      MD311 AT %MD311 : UDINT := 16#00000000;  (* RAD[1].Fk: Площадь конвекции *)
      MD312 AT %MD312 : UDINT := 16#00000000;  (* RAD[1].Q0: Расход своб конвекции *)
      MD313 AT %MD313 : UDINT := 16#00000000;  (* RAD[1].Q1: Расход принуд конвекции *)
      MD314 AT %MD314 : UDINT := 16#00000000;  (* RAD[1].Bl[0]: Vобдува- 1 вентилятор *)
      MD315 AT %MD315 : UDINT := 16#00000000;  (* RAD[1].Bl[1]: Vобдува- 2 вентилятора *)
      MD316 AT %MD316 : UDINT := 16#00000000;  (* RAD[1].Bl[2]: Vобдува- 3 вентилятора *)
      MD317 AT %MD317 : UDINT := 16#00000000;  (* RAD[1].Bl[3]: Vобдува- 4 вентилятора *)
      MD318 AT %MD318 : UDINT := 16#00000000;  (* RAD[2].Vm: Объем радиатора *)
      MD319 AT %MD319 : UDINT := 16#00000000;  (* RAD[2].Fk: Площадь конвекции *)
      MD320 AT %MD320 : UDINT := 16#00000000;  (* RAD[2].Q0: Расход своб конвекции *)
      MD321 AT %MD321 : UDINT := 16#00000000;  (* RAD[2].Q1: Расход принуд конвекции *)
      MD322 AT %MD322 : UDINT := 16#00000000;  (* RAD[2].Bl[0]: Vобдува- 1 вентилятор *)
      MD323 AT %MD323 : UDINT := 16#00000000;  (* RAD[2].Bl[1]: Vобдува- 2 вентилятора *)
      MD324 AT %MD324 : UDINT := 16#00000000;  (* RAD[2].Bl[2]: Vобдува- 3 вентилятора *)
      MD325 AT %MD325 : UDINT := 16#00000000;  (* RAD[2].Bl[3]: Vобдува- 4 вентилятора *)
      MD326 AT %MD326 : UDINT := 16#00000000;  (* RAD[3].Vm: Объем радиатора *)
      MD327 AT %MD327 : UDINT := 16#00000000;  (* RAD[3].Fk: Площадь конвекции *)
      MD328 AT %MD328 : UDINT := 16#00000000;  (* RAD[3].Q0: Расход своб конвекции *)
      MD329 AT %MD329 : UDINT := 16#00000000;  (* RAD[3].Q1: Расход принуд конвекции *)
      MD330 AT %MD330 : UDINT := 16#00000000;  (* RAD[3].Bl[0]: Vобдува- 1 вентилятор *)
      MD331 AT %MD331 : UDINT := 16#00000000;  (* RAD[3].Bl[1]: Vобдува- 2 вентилятора *)
      MD332 AT %MD332 : UDINT := 16#00000000;  (* RAD[3].Bl[2]: Vобдува- 3 вентилятора *)
      MD333 AT %MD333 : UDINT := 16#00000000;  (* RAD[3].Bl[3]: Vобдува- 4 вентилятора *)
      MD334 AT %MD334 : UDINT := 16#00000000;  (* RAD[4].Vm: Объем радиатора *)
      MD335 AT %MD335 : UDINT := 16#00000000;  (* RAD[4].Fk: Площадь конвекции *)
      MD336 AT %MD336 : UDINT := 16#00000000;  (* RAD[4].Q0: Расход своб конвекции *)
      MD337 AT %MD337 : UDINT := 16#00000000;  (* RAD[4].Q1: Расход принуд конвекции *)
      MD338 AT %MD338 : UDINT := 16#00000000;  (* RAD[4].Bl[0]: Vобдува- 1 вентилятор *)
      MD339 AT %MD339 : UDINT := 16#00000000;  (* RAD[4].Bl[1]: Vобдува- 2 вентилятора *)
      MD340 AT %MD340 : UDINT := 16#00000000;  (* RAD[4].Bl[2]: Vобдува- 3 вентилятора *)
      MD341 AT %MD341 : UDINT := 16#00000000;  (* RAD[4].Bl[3]: Vобдува- 4 вентилятора *)
      MD342 AT %MD342 : UDINT := 16#00000000;  (* RAD[5].Vm: Объем радиатора *)
      MD343 AT %MD343 : UDINT := 16#00000000;  (* RAD[5].Fk: Площадь конвекции *)
      MD344 AT %MD344 : UDINT := 16#00000000;  (* RAD[5].Q0: Расход своб конвекции *)
      MD345 AT %MD345 : UDINT := 16#00000000;  (* RAD[5].Q1: Расход принуд конвекции *)
      MD346 AT %MD346 : UDINT := 16#00000000;  (* RAD[5].Bl[0]: Vобдува- 1 вентилятор *)
      MD347 AT %MD347 : UDINT := 16#00000000;  (* RAD[5].Bl[1]: Vобдува- 2 вентилятора *)
      MD348 AT %MD348 : UDINT := 16#00000000;  (* RAD[5].Bl[2]: Vобдува- 3 вентилятора *)
      MD349 AT %MD349 : UDINT := 16#00000000;  (* RAD[5].Bl[3]: Vобдува- 4 вентилятора *)
      MD350 AT %MD350 : UDINT := 16#00000000;  (* RAD[6].Vm: Объем радиатора *)
      MD351 AT %MD351 : UDINT := 16#00000000;  (* RAD[6].Fk: Площадь конвекции *)
      MD352 AT %MD352 : UDINT := 16#00000000;  (* RAD[6].Q0: Расход своб конвекции *)
      MD353 AT %MD353 : UDINT := 16#00000000;  (* RAD[6].Q1: Расход принуд конвекции *)
      MD354 AT %MD354 : UDINT := 16#00000000;  (* RAD[6].Bl[0]: Vобдува- 1 вентилятор *)
      MD355 AT %MD355 : UDINT := 16#00000000;  (* RAD[6].Bl[1]: Vобдува- 2 вентилятора *)
      MD356 AT %MD356 : UDINT := 16#00000000;  (* RAD[6].Bl[2]: Vобдува- 3 вентилятора *)
      MD357 AT %MD357 : UDINT := 16#00000000;  (* RAD[6].Bl[3]: Vобдува- 4 вентилятора *)
      MD358 AT %MD358 : UDINT := 16#00000000;  (* RAD[7].Vm: Объем радиатора *)
      MD359 AT %MD359 : UDINT := 16#00000000;  (* RAD[7].Fk: Площадь конвекции *)
      MD360 AT %MD360 : UDINT := 16#00000000;  (* RAD[7].Q0: Расход своб конвекции *)
      MD361 AT %MD361 : UDINT := 16#00000000;  (* RAD[7].Q1: Расход принуд конвекции *)
      MD362 AT %MD362 : UDINT := 16#00000000;  (* RAD[7].Bl[0]: Vобдува- 1 вентилятор *)
      MD363 AT %MD363 : UDINT := 16#00000000;  (* RAD[7].Bl[1]: Vобдува- 2 вентилятора *)
      MD364 AT %MD364 : UDINT := 16#00000000;  (* RAD[7].Bl[2]: Vобдува- 3 вентилятора *)
      MD365 AT %MD365 : UDINT := 16#00000000;  (* RAD[7].Bl[3]: Vобдува- 4 вентилятора *)
      MD366 AT %MD366 : UDINT := 16#00000000;  (* RAD[8].Vm: Объем радиатора *)
      MD367 AT %MD367 : UDINT := 16#00000000;  (* RAD[8].Fk: Площадь конвекции *)
      MD368 AT %MD368 : UDINT := 16#00000000;  (* RAD[8].Q0: Расход своб конвекции *)
      MD369 AT %MD369 : UDINT := 16#00000000;  (* RAD[8].Q1: Расход принуд конвекции *)
      MD370 AT %MD370 : UDINT := 16#00000000;  (* RAD[8].Bl[0]: Vобдува- 1 вентилятор *)
      MD371 AT %MD371 : UDINT := 16#00000000;  (* RAD[8].Bl[1]: Vобдува- 2 вентилятора *)
      MD372 AT %MD372 : UDINT := 16#00000000;  (* RAD[8].Bl[2]: Vобдува- 3 вентилятора *)
      MD373 AT %MD373 : UDINT := 16#00000000;  (* RAD[8].Bl[3]: Vобдува- 4 вентилятора *)
      MD374 AT %MD374 : UDINT := 16#00000000;  (* RAD[9].Vm: Объем радиатора *)
      MD375 AT %MD375 : UDINT := 16#00000000;  (* RAD[9].Fk: Площадь конвекции *)
      MD376 AT %MD376 : UDINT := 16#00000000;  (* RAD[9].Q0: Расход своб конвекции *)
      MD377 AT %MD377 : UDINT := 16#00000000;  (* RAD[9].Q1: Расход принуд конвекции *)
      MD378 AT %MD378 : UDINT := 16#00000000;  (* RAD[9].Bl[0]: Vобдува- 1 вентилятор *)
      MD379 AT %MD379 : UDINT := 16#00000000;  (* RAD[9].Bl[1]: Vобдува- 2 вентилятора *)
      MD380 AT %MD380 : UDINT := 16#00000000;  (* RAD[9].Bl[2]: Vобдува- 3 вентилятора *)
      MD381 AT %MD381 : UDINT := 16#00000000;  (* RAD[9].Bl[3]: Vобдува- 4 вентилятора *)
      MD382 AT %MD382 : UDINT := 16#00000000;  (* RAD[10].Vm: Объем радиатора *)
      MD383 AT %MD383 : UDINT := 16#00000000;  (* RAD[10].Fk: Площадь конвекции *)
      MD384 AT %MD384 : UDINT := 16#00000000;  (* RAD[10].Q0: Расход своб конвекции *)
      MD385 AT %MD385 : UDINT := 16#00000000;  (* RAD[10].Q1: Расход принуд конвекции *)
      MD386 AT %MD386 : UDINT := 16#00000000;  (* RAD[10].Bl[0]: Vобдува- 1 вентилятор *)
      MD387 AT %MD387 : UDINT := 16#00000000;  (* RAD[10].Bl[1]: Vобдува- 2 вентилятора *)
      MD388 AT %MD388 : UDINT := 16#00000000;  (* RAD[10].Bl[2]: Vобдува- 3 вентилятора *)
      MD389 AT %MD389 : UDINT := 16#00000000;  (* RAD[10].Bl[3]: Vобдува- 4 вентилятора *)
      MD390 AT %MD390 : UDINT := 16#00000000;  (* RAD[11].Vm: Объем радиатора *)
      MD391 AT %MD391 : UDINT := 16#00000000;  (* RAD[11].Fk: Площадь конвекции *)
      MD392 AT %MD392 : UDINT := 16#00000000;  (* RAD[11].Q0: Расход своб конвекции *)
      MD393 AT %MD393 : UDINT := 16#00000000;  (* RAD[11].Q1: Расход принуд конвекции *)
      MD394 AT %MD394 : UDINT := 16#00000000;  (* RAD[11].Bl[0]: Vобдува- 1 вентилятор *)
      MD395 AT %MD395 : UDINT := 16#00000000;  (* RAD[11].Bl[1]: Vобдува- 2 вентилятора *)
      MD396 AT %MD396 : UDINT := 16#00000000;  (* RAD[11].Bl[2]: Vобдува- 3 вентилятора *)
      MD397 AT %MD397 : UDINT := 16#00000000;  (* RAD[11].Bl[3]: Vобдува- 4 вентилятора *)
      MD398 AT %MD398 : UDINT := 16#00000000;  (* RAD[12].Vm: Объем радиатора *)
      MD399 AT %MD399 : UDINT := 16#00000000;  (* RAD[12].Fk: Площадь конвекции *)
      MD400 AT %MD400 : UDINT := 16#00000000;  (* RAD[12].Q0: Расход своб конвекции *)
      MD401 AT %MD401 : UDINT := 16#00000000;  (* RAD[12].Q1: Расход принуд конвекции *)
      MD402 AT %MD402 : UDINT := 16#00000000;  (* RAD[12].Bl[0]: Vобдува- 1 вентилятор *)
      MD403 AT %MD403 : UDINT := 16#00000000;  (* RAD[12].Bl[1]: Vобдува- 2 вентилятора *)
      MD404 AT %MD404 : UDINT := 16#00000000;  (* RAD[12].Bl[2]: Vобдува- 3 вентилятора *)
      MD405 AT %MD405 : UDINT := 16#00000000;  (* RAD[12].Bl[3]: Vобдува- 4 вентилятора *)
      MD406 AT %MD406 : UDINT := 16#00000000;  (* RAD[13].Vm: Объем радиатора *)
      MD407 AT %MD407 : UDINT := 16#00000000;  (* RAD[13].Fk: Площадь конвекции *)
      MD408 AT %MD408 : UDINT := 16#00000000;  (* RAD[13].Q0: Расход своб конвекции *)
      MD409 AT %MD409 : UDINT := 16#00000000;  (* RAD[13].Q1: Расход принуд конвекции *)
      MD410 AT %MD410 : UDINT := 16#00000000;  (* RAD[13].Bl[0]: Vобдува- 1 вентилятор *)
      MD411 AT %MD411 : UDINT := 16#00000000;  (* RAD[13].Bl[1]: Vобдува- 2 вентилятора *)
      MD412 AT %MD412 : UDINT := 16#00000000;  (* RAD[13].Bl[2]: Vобдува- 3 вентилятора *)
      MD413 AT %MD413 : UDINT := 16#00000000;  (* RAD[13].Bl[3]: Vобдува- 4 вентилятора *)
      MD414 AT %MD414 : UDINT := 16#00000000;  (* RAD[14].Vm: Объем радиатора *)
      MD415 AT %MD415 : UDINT := 16#00000000;  (* RAD[14].Fk: Площадь конвекции *)
      MD416 AT %MD416 : UDINT := 16#00000000;  (* RAD[14].Q0: Расход своб конвекции *)
      MD417 AT %MD417 : UDINT := 16#00000000;  (* RAD[14].Q1: Расход принуд конвекции *)
      MD418 AT %MD418 : UDINT := 16#00000000;  (* RAD[14].Bl[0]: Vобдува- 1 вентилятор *)
      MD419 AT %MD419 : UDINT := 16#00000000;  (* RAD[14].Bl[1]: Vобдува- 2 вентилятора *)
      MD420 AT %MD420 : UDINT := 16#00000000;  (* RAD[14].Bl[2]: Vобдува- 3 вентилятора *)
      MD421 AT %MD421 : UDINT := 16#00000000;  (* RAD[14].Bl[3]: Vобдува- 4 вентилятора *)
      MD422 AT %MD422 : UDINT := 16#00000000;  (* RAD[15].Vm: Объем радиатора *)
      MD423 AT %MD423 : UDINT := 16#00000000;  (* RAD[15].Fk: Площадь конвекции *)
      MD424 AT %MD424 : UDINT := 16#00000000;  (* RAD[15].Q0: Расход своб конвекции *)
      MD425 AT %MD425 : UDINT := 16#00000000;  (* RAD[15].Q1: Расход принуд конвекции *)
      MD426 AT %MD426 : UDINT := 16#00000000;  (* RAD[15].Bl[0]: Vобдува- 1 вентилятор *)
      MD427 AT %MD427 : UDINT := 16#00000000;  (* RAD[15].Bl[1]: Vобдува- 2 вентилятора *)
      MD428 AT %MD428 : UDINT := 16#00000000;  (* RAD[15].Bl[2]: Vобдува- 3 вентилятора *)
      MD429 AT %MD429 : UDINT := 16#00000000;  (* RAD[15].Bl[3]: Vобдува- 4 вентилятора *)
      MD430 AT %MD430 : UDINT := 16#00000000;  (* HDI.DTI: Дата (секунд от 1970-01-01) *)
      MD431 AT %MD431 : UDINT := 16#00000000;  (* HDI.TMI: Время (милисек с 00:00) *)
      MD432 AT %MD432 : UDINT := 16#00000000;  (* HDI.TOV: Темп. окр. воздуха *)
      MD433 AT %MD433 : UDINT := 16#00000000;  (* HDI.TMH: Темп. верх. слоёв масла *)
      MD434 AT %MD434 : UDINT := 16#00000000;  (* HDI.RVI[0]: Резерв 0 *)
      MD435 AT %MD435 : UDINT := 16#00000000;  (* HDI.RVI[1]: Резерв 1 *)
      MD436 AT %MD436 : UDINT := 16#00000000;  (* PHI[0].Ic: Ток нагрузки *)
      MD437 AT %MD437 : UDINT := 16#00000000;  (* PHI[0].Tin: Т входа из сист.охл. *)
      MD438 AT %MD438 : UDINT := 16#00000000;  (* PHI[0].Tout: Т выхода из сист.охл. *)
      MD439 AT %MD439 : UDINT := 16#00000000;  (* PHI[0].Rn: 32-бит состояния РПН *)
      MD440 AT %MD440 : UDINT := 16#00000000;  (* PHI[0].RD[0,1]: Радиатор-0,1: Тип-Состояние *)
      MD441 AT %MD441 : UDINT := 16#00000000;  (* PHI[0].RD[2,3]: Радиатор-2,3: Тип-Состояние *)
      MD442 AT %MD442 : UDINT := 16#00000000;  (* PHI[0].RD[4,5]: Радиатор-4,5: Тип-Состояние *)
      MD443 AT %MD443 : UDINT := 16#00000000;  (* PHI[0].RD[6,7]: Радиатор-6,7: Тип-Состояние *)
      MD444 AT %MD444 : UDINT := 16#00000000;  (* PHI[1].Ic: Ток нагрузки *)
      MD445 AT %MD445 : UDINT := 16#00000000;  (* PHI[1].Tin: Т входа из сист.охл. *)
      MD446 AT %MD446 : UDINT := 16#00000000;  (* PHI[1].Tout: Т выхода из сист.охл. *)
      MD447 AT %MD447 : UDINT := 16#00000000;  (* PHI[1].Rn: 32-бит состояния РПН *)
      MD448 AT %MD448 : UDINT := 16#00000000;  (* PHI[1].RD[0,1]: Радиатор-0,1: Тип-Состояние *)
      MD449 AT %MD449 : UDINT := 16#00000000;  (* PHI[1].RD[2,3]: Радиатор-2,3: Тип-Состояние *)
      MD450 AT %MD450 : UDINT := 16#00000000;  (* PHI[1].RD[4,5]: Радиатор-4,5: Тип-Состояние *)
      MD451 AT %MD451 : UDINT := 16#00000000;  (* PHI[1].RD[6,7]: Радиатор-6,7: Тип-Состояние *)
      MD452 AT %MD452 : UDINT := 16#00000000;  (* PHI[2].Ic: Ток нагрузки *)
      MD453 AT %MD453 : UDINT := 16#00000000;  (* PHI[2].Tin: Т входа из сист.охл. *)
      MD454 AT %MD454 : UDINT := 16#00000000;  (* PHI[2].Tout: Т выхода из сист.охл. *)
      MD455 AT %MD455 : UDINT := 16#00000000;  (* PHI[2].Rn: 32-бит состояния РПН *)
      MD456 AT %MD456 : UDINT := 16#00000000;  (* PHI[2].RD[0,1]: Радиатор-0,1: Тип-Состояние *)
      MD457 AT %MD457 : UDINT := 16#00000000;  (* PHI[2].RD[2,3]: Радиатор-2,3: Тип-Состояние *)
      MD458 AT %MD458 : UDINT := 16#00000000;  (* PHI[2].RD[4,5]: Радиатор-4,5: Тип-Состояние *)
      MD459 AT %MD459 : UDINT := 16#00000000;  (* PHI[2].RD[6,7]: Радиатор-6,7: Тип-Состояние *)
      MD460 AT %MD460 : UDINT := 16#00000000;  (* HDO.DTO: Дата (секунд от 1970-01-01) *)
      MD461 AT %MD461 : UDINT := 16#00000000;  (* HDO.TMO: Время (милисек с 00:00) *)
      MD462 AT %MD462 : UDINT := 16#00000000;  (* HDO.QTY: Плотность потока ярма *)
      MD463 AT %MD463 : UDINT := 16#00000000;  (* HDO.QTS: Общее тепловыделение *)
      MD464 AT %MD464 : UDINT := 16#00000000;  (* HDO.RVO[0]: Резерв 0 *)
      MD465 AT %MD465 : UDINT := 16#00000000;  (* HDO.RVO[1]: Резерв 1 *)
      MD466 AT %MD466 : UDINT := 16#00000000;  (* PHO[0].Q0: Плотность потока стержня *)
      MD467 AT %MD467 : UDINT := 16#00000000;  (* PHO[0].Q1: Плотность потока обмотки НН *)
      MD468 AT %MD468 : UDINT := 16#00000000;  (* PHO[0].Q2: Плотность потока обмотки ВН *)
      MD469 AT %MD469 : UDINT := 16#00000000;  (* PHO[0].Tin: Т входа из сист.охл. *)
      MD470 AT %MD470 : UDINT := 16#00000000;  (* PHO[0].Tout: Т выхода из сист.охл. *)
      MD471 AT %MD471 : UDINT := 16#00000000;  (* PHO[0].Qm: Суммарный расход масла на фазу *)
      MD472 AT %MD472 : UDINT := 16#00000000;  (* PHO[0].Se: Экв площадь сечения каналов *)
      MD473 AT %MD473 : UDINT := 16#00000000;  (* PHO[0].Ve: Скорость тока масла на фазу *)
      MD474 AT %MD474 : UDINT := 16#00000000;  (* PHO[1].Q0: Плотность потока стержня *)
      MD475 AT %MD475 : UDINT := 16#00000000;  (* PHO[1].Q1: Плотность потока обмотки НН *)
      MD476 AT %MD476 : UDINT := 16#00000000;  (* PHO[1].Q2: Плотность потока обмотки ВН *)
      MD477 AT %MD477 : UDINT := 16#00000000;  (* PHO[1].Tin: Т входа из сист.охл. *)
      MD478 AT %MD478 : UDINT := 16#00000000;  (* PHO[1].Tout: Т выхода из сист.охл. *)
      MD479 AT %MD479 : UDINT := 16#00000000;  (* PHO[1].Qm: Суммарный расход масла на фазу *)
      MD480 AT %MD480 : UDINT := 16#00000000;  (* PHO[1].Se: Экв площадь сечения каналов *)
      MD481 AT %MD481 : UDINT := 16#00000000;  (* PHO[1].Ve: Скорость тока масла на фазу *)
      MD482 AT %MD482 : UDINT := 16#00000000;  (* PHO[2].Q0: Плотность потока стержня *)
      MD483 AT %MD483 : UDINT := 16#00000000;  (* PHO[2].Q1: Плотность потока обмотки НН *)
      MD484 AT %MD484 : UDINT := 16#00000000;  (* PHO[2].Q2: Плотность потока обмотки ВН *)
      MD485 AT %MD485 : UDINT := 16#00000000;  (* PHO[2].Tin: Т входа из сист.охл. *)
      MD486 AT %MD486 : UDINT := 16#00000000;  (* PHO[2].Tout: Т выхода из сист.охл. *)
      MD487 AT %MD487 : UDINT := 16#00000000;  (* PHO[2].Qm: Суммарный расход масла на фазу *)
      MD488 AT %MD488 : UDINT := 16#00000000;  (* PHO[2].Se: Экв площадь сечения каналов *)
      MD489 AT %MD489 : UDINT := 16#00000000;  (* PHO[2].Ve: Скорость тока масла на фазу *)
      MD490 AT %MD490 : UDINT := 16#00000000;  (* RES.DR: Дата (секунд от 1970-01-01) *)
      MD491 AT %MD491 : UDINT := 16#00000000;  (* RES.TR: Время (милисек с 00:00) *)
      MD492 AT %MD492 : UDINT := 16#00000000;  (* RES.FP: Факт. время расчёта (милисек) *)
      MD493 AT %MD493 : UDINT := 16#00000000;  (* RES.ER|RES.FL: Ошибка(UINT)|Флаги(WORD) *)
      MD494 AT %MD494 : UDINT := 16#00000000;  (* RES.RD[0]: Резерв 0 *)
      MD495 AT %MD495 : UDINT := 16#00000000;  (* RES.RD[1]: Резерв 1 *)
      MD496 AT %MD496 : UDINT := 16#00000000;  (* RES.RD[2]: Резерв 2 *)
      MD497 AT %MD497 : UDINT := 16#00000000;  (* RES.RD[3]: Резерв 3 *)
      MD498 AT %MD498 : UDINT := 16#00000000;  (* RES.RD[4]: Резерв 4 *)
      MD499 AT %MD499 : UDINT := 16#00000000;  (* RES.RD[5]: Резерв 5 *)
      MD500 AT %MD500 : UDINT := 16#00000000;  (* CDN[0].(ID|Tmid): Идент.|Tсред. *)
      MD501 AT %MD501 : UDINT := 16#00000000;  (* CDN[0].Tmin.(Ti |XYZ[0]): Темп. |Коорд.X *)
      MD502 AT %MD502 : UDINT := 16#00000000;  (* CDN[0].Tmin.(XYZ[1]|XYZ[2]): Коорд.Y|Коорд.Z *)
      MD503 AT %MD503 : UDINT := 16#00000000;  (* CDN[0].Tmax.(Ti |XYZ[0]): Темп. |Коорд.X *)
      MD504 AT %MD504 : UDINT := 16#00000000;  (* CDN[0].Tmax.(XYZ[1]|XYZ[2]): Коорд.Y|Коорд.Z *)
      MD505 AT %MD505 : UDINT := 16#00000000;  (* CDN[1].(ID|Tmid): Идент.|Tсред. *)
      MD506 AT %MD506 : UDINT := 16#00000000;  (* CDN[1].Tmin.(Ti |XYZ[0]): Темп. |Коорд.X *)
      MD507 AT %MD507 : UDINT := 16#00000000;  (* CDN[1].Tmin.(XYZ[1]|XYZ[2]): Коорд.Y|Коорд.Z *)
      MD508 AT %MD508 : UDINT := 16#00000000;  (* CDN[1].Tmax.(Ti |XYZ[0]): Темп. |Коорд.X *)
      MD509 AT %MD509 : UDINT := 16#00000000;  (* CDN[1].Tmax.(XYZ[1]|XYZ[2]): Коорд.Y|Коорд.Z *)
      MD510 AT %MD510 : UDINT := 16#00000000;  (* CDN[2].(ID|Tmid): Идент.|Tсред. *)
      MD511 AT %MD511 : UDINT := 16#00000000;  (* CDN[2].Tmin.(Ti |XYZ[0]): Темп. |Коорд.X *)
      MD512 AT %MD512 : UDINT := 16#00000000;  (* CDN[2].Tmin.(XYZ[1]|XYZ[2]): Коорд.Y|Коорд.Z *)
      MD513 AT %MD513 : UDINT := 16#00000000;  (* CDN[2].Tmax.(Ti |XYZ[0]): Темп. |Коорд.X *)
      MD514 AT %MD514 : UDINT := 16#00000000;  (* CDN[2].Tmax.(XYZ[1]|XYZ[2]): Коорд.Y|Коорд.Z *)
      MD515 AT %MD515 : UDINT := 16#00000000;  (* CDN[3].(ID|Tmid): Идент.|Tсред. *)
      MD516 AT %MD516 : UDINT := 16#00000000;  (* CDN[3].Tmin.(Ti |XYZ[0]): Темп. |Коорд.X *)
      MD517 AT %MD517 : UDINT := 16#00000000;  (* CDN[3].Tmin.(XYZ[1]|XYZ[2]): Коорд.Y|Коорд.Z *)
      MD518 AT %MD518 : UDINT := 16#00000000;  (* CDN[3].Tmax.(Ti |XYZ[0]): Темп. |Коорд.X *)
      MD519 AT %MD519 : UDINT := 16#00000000;  (* CDN[3].Tmax.(XYZ[1]|XYZ[2]): Коорд.Y|Коорд.Z *)
      MD520 AT %MD520 : UDINT := 16#00000000;  (* CDN[4].(ID|Tmid): Идент.|Tсред. *)
      MD521 AT %MD521 : UDINT := 16#00000000;  (* CDN[4].Tmin.(Ti |XYZ[0]): Темп. |Коорд.X *)
      MD522 AT %MD522 : UDINT := 16#00000000;  (* CDN[4].Tmin.(XYZ[1]|XYZ[2]): Коорд.Y|Коорд.Z *)
      MD523 AT %MD523 : UDINT := 16#00000000;  (* CDN[4].Tmax.(Ti |XYZ[0]): Темп. |Коорд.X *)
      MD524 AT %MD524 : UDINT := 16#00000000;  (* CDN[4].Tmax.(XYZ[1]|XYZ[2]): Коорд.Y|Коорд.Z *)
      MD525 AT %MD525 : UDINT := 16#00000000;  (* CDN[5].(ID|Tmid): Идент.|Tсред. *)
      MD526 AT %MD526 : UDINT := 16#00000000;  (* CDN[5].Tmin.(Ti |XYZ[0]): Темп. |Коорд.X *)
      MD527 AT %MD527 : UDINT := 16#00000000;  (* CDN[5].Tmin.(XYZ[1]|XYZ[2]): Коорд.Y|Коорд.Z *)
      MD528 AT %MD528 : UDINT := 16#00000000;  (* CDN[5].Tmax.(Ti |XYZ[0]): Темп. |Коорд.X *)
      MD529 AT %MD529 : UDINT := 16#00000000;  (* CDN[5].Tmax.(XYZ[1]|XYZ[2]): Коорд.Y|Коорд.Z *)
      MD530 AT %MD530 : UDINT := 16#00000000;  (* CDN[6].(ID|Tmid): Идент.|Tсред. *)
      MD531 AT %MD531 : UDINT := 16#00000000;  (* CDN[6].Tmin.(Ti |XYZ[0]): Темп. |Коорд.X *)
      MD532 AT %MD532 : UDINT := 16#00000000;  (* CDN[6].Tmin.(XYZ[1]|XYZ[2]): Коорд.Y|Коорд.Z *)
      MD533 AT %MD533 : UDINT := 16#00000000;  (* CDN[6].Tmax.(Ti |XYZ[0]): Темп. |Коорд.X *)
      MD534 AT %MD534 : UDINT := 16#00000000;  (* CDN[6].Tmax.(XYZ[1]|XYZ[2]): Коорд.Y|Коорд.Z *)
      MD535 AT %MD535 : UDINT := 16#00000000;  (* CDN[7].(ID|Tmid): Идент.|Tсред. *)
      MD536 AT %MD536 : UDINT := 16#00000000;  (* CDN[7].Tmin.(Ti |XYZ[0]): Темп. |Коорд.X *)
      MD537 AT %MD537 : UDINT := 16#00000000;  (* CDN[7].Tmin.(XYZ[1]|XYZ[2]): Коорд.Y|Коорд.Z *)
      MD538 AT %MD538 : UDINT := 16#00000000;  (* CDN[7].Tmax.(Ti |XYZ[0]): Темп. |Коорд.X *)
      MD539 AT %MD539 : UDINT := 16#00000000;  (* CDN[7].Tmax.(XYZ[1]|XYZ[2]): Коорд.Y|Коорд.Z *)
      MD540 AT %MD540 : UDINT := 16#00000000;  (* CDN[8].(ID|Tmid): Идент.|Tсред. *)
      MD541 AT %MD541 : UDINT := 16#00000000;  (* CDN[8].Tmin.(Ti |XYZ[0]): Темп. |Коорд.X *)
      MD542 AT %MD542 : UDINT := 16#00000000;  (* CDN[8].Tmin.(XYZ[1]|XYZ[2]): Коорд.Y|Коорд.Z *)
      MD543 AT %MD543 : UDINT := 16#00000000;  (* CDN[8].Tmax.(Ti |XYZ[0]): Темп. |Коорд.X *)
      MD544 AT %MD544 : UDINT := 16#00000000;  (* CDN[8].Tmax.(XYZ[1]|XYZ[2]): Коорд.Y|Коорд.Z *)
      MD545 AT %MD545 : UDINT := 16#00000000;  (* CDN[9].(ID|Tmid): Идент.|Tсред. *)
      MD546 AT %MD546 : UDINT := 16#00000000;  (* CDN[9].Tmin.(Ti |XYZ[0]): Темп. |Коорд.X *)
      MD547 AT %MD547 : UDINT := 16#00000000;  (* CDN[9].Tmin.(XYZ[1]|XYZ[2]): Коорд.Y|Коорд.Z *)
      MD548 AT %MD548 : UDINT := 16#00000000;  (* CDN[9].Tmax.(Ti |XYZ[0]): Темп. |Коорд.X *)
      MD549 AT %MD549 : UDINT := 16#00000000;  (* CDN[9].Tmax.(XYZ[1]|XYZ[2]): Коорд.Y|Коорд.Z *)
      MD550 AT %MD550 : UDINT := 16#00000000;  (* CDN[10].(ID|Tmid): Идент.|Tсред. *)
      MD551 AT %MD551 : UDINT := 16#00000000;  (* CDN[10].Tmin.(Ti |XYZ[0]): Темп. |Коорд.X *)
      MD552 AT %MD552 : UDINT := 16#00000000;  (* CDN[10].Tmin.(XYZ[1]|XYZ[2]): Коорд.Y|Коорд.Z *)
      MD553 AT %MD553 : UDINT := 16#00000000;  (* CDN[10].Tmax.(Ti |XYZ[0]): Темп. |Коорд.X *)
      MD554 AT %MD554 : UDINT := 16#00000000;  (* CDN[10].Tmax.(XYZ[1]|XYZ[2]): Коорд.Y|Коорд.Z *)
      MD555 AT %MD555 : UDINT := 16#00000000;  (* CDN[11].(ID|Tmid): Идент.|Tсред. *)
      MD556 AT %MD556 : UDINT := 16#00000000;  (* CDN[11].Tmin.(Ti |XYZ[0]): Темп. |Коорд.X *)
      MD557 AT %MD557 : UDINT := 16#00000000;  (* CDN[11].Tmin.(XYZ[1]|XYZ[2]): Коорд.Y|Коорд.Z *)
      MD558 AT %MD558 : UDINT := 16#00000000;  (* CDN[11].Tmax.(Ti |XYZ[0]): Темп. |Коорд.X *)
      MD559 AT %MD559 : UDINT := 16#00000000;  (* CDN[11].Tmax.(XYZ[1]|XYZ[2]): Коорд.Y|Коорд.Z *)
      MD560 AT %MD560 : UDINT := 16#00000000;  (* CDN[12].(ID|Tmid): Идент.|Tсред. *)
      MD561 AT %MD561 : UDINT := 16#00000000;  (* CDN[12].Tmin.(Ti |XYZ[0]): Темп. |Коорд.X *)
      MD562 AT %MD562 : UDINT := 16#00000000;  (* CDN[12].Tmin.(XYZ[1]|XYZ[2]): Коорд.Y|Коорд.Z *)
      MD563 AT %MD563 : UDINT := 16#00000000;  (* CDN[12].Tmax.(Ti |XYZ[0]): Темп. |Коорд.X *)
      MD564 AT %MD564 : UDINT := 16#00000000;  (* CDN[12].Tmax.(XYZ[1]|XYZ[2]): Коорд.Y|Коорд.Z *)
      MD565 AT %MD565 : UDINT := 16#00000000;  (* CDN[13].(ID|Tmid): Идент.|Tсред. *)
      MD566 AT %MD566 : UDINT := 16#00000000;  (* CDN[13].Tmin.(Ti |XYZ[0]): Темп. |Коорд.X *)
      MD567 AT %MD567 : UDINT := 16#00000000;  (* CDN[13].Tmin.(XYZ[1]|XYZ[2]): Коорд.Y|Коорд.Z *)
      MD568 AT %MD568 : UDINT := 16#00000000;  (* CDN[13].Tmax.(Ti |XYZ[0]): Темп. |Коорд.X *)
      MD569 AT %MD569 : UDINT := 16#00000000;  (* CDN[13].Tmax.(XYZ[1]|XYZ[2]): Коорд.Y|Коорд.Z *)
      MD570 AT %MD570 : UDINT := 16#00000000;  (* CDN[14].(ID|Tmid): Идент.|Tсред. *)
      MD571 AT %MD571 : UDINT := 16#00000000;  (* CDN[14].Tmin.(Ti |XYZ[0]): Темп. |Коорд.X *)
      MD572 AT %MD572 : UDINT := 16#00000000;  (* CDN[14].Tmin.(XYZ[1]|XYZ[2]): Коорд.Y|Коорд.Z *)
      MD573 AT %MD573 : UDINT := 16#00000000;  (* CDN[14].Tmax.(Ti |XYZ[0]): Темп. |Коорд.X *)
      MD574 AT %MD574 : UDINT := 16#00000000;  (* CDN[14].Tmax.(XYZ[1]|XYZ[2]): Коорд.Y|Коорд.Z *)
      MD575 AT %MD575 : UDINT := 16#00000000;  (* CDN[15].(ID|Tmid): Идент.|Tсред. *)
      MD576 AT %MD576 : UDINT := 16#00000000;  (* CDN[15].Tmin.(Ti |XYZ[0]): Темп. |Коорд.X *)
      MD577 AT %MD577 : UDINT := 16#00000000;  (* CDN[15].Tmin.(XYZ[1]|XYZ[2]): Коорд.Y|Коорд.Z *)
      MD578 AT %MD578 : UDINT := 16#00000000;  (* CDN[15].Tmax.(Ti |XYZ[0]): Темп. |Коорд.X *)
      MD579 AT %MD579 : UDINT := 16#00000000;  (* CDN[15].Tmax.(XYZ[1]|XYZ[2]): Коорд.Y|Коорд.Z *)
      MD580 AT %MD580 : UDINT := 16#00000000;  (* CDN[16].(ID|Tmid): Идент.|Tсред. *)
      MD581 AT %MD581 : UDINT := 16#00000000;  (* CDN[16].Tmin.(Ti |XYZ[0]): Темп. |Коорд.X *)
      MD582 AT %MD582 : UDINT := 16#00000000;  (* CDN[16].Tmin.(XYZ[1]|XYZ[2]): Коорд.Y|Коорд.Z *)
      MD583 AT %MD583 : UDINT := 16#00000000;  (* CDN[16].Tmax.(Ti |XYZ[0]): Темп. |Коорд.X *)
      MD584 AT %MD584 : UDINT := 16#00000000;  (* CDN[16].Tmax.(XYZ[1]|XYZ[2]): Коорд.Y|Коорд.Z *)
      MD585 AT %MD585 : UDINT := 16#00000000;  (* CDN[17].(ID|Tmid): Идент.|Tсред. *)
      MD586 AT %MD586 : UDINT := 16#00000000;  (* CDN[17].Tmin.(Ti |XYZ[0]): Темп. |Коорд.X *)
      MD587 AT %MD587 : UDINT := 16#00000000;  (* CDN[17].Tmin.(XYZ[1]|XYZ[2]): Коорд.Y|Коорд.Z *)
      MD588 AT %MD588 : UDINT := 16#00000000;  (* CDN[17].Tmax.(Ti |XYZ[0]): Темп. |Коорд.X *)
      MD589 AT %MD589 : UDINT := 16#00000000;  (* CDN[17].Tmax.(XYZ[1]|XYZ[2]): Коорд.Y|Коорд.Z *)
      MD590 AT %MD590 : UDINT := 16#00000000;  (* CDN[18].(ID|Tmid): Идент.|Tсред. *)
      MD591 AT %MD591 : UDINT := 16#00000000;  (* CDN[18].Tmin.(Ti |XYZ[0]): Темп. |Коорд.X *)
      MD592 AT %MD592 : UDINT := 16#00000000;  (* CDN[18].Tmin.(XYZ[1]|XYZ[2]): Коорд.Y|Коорд.Z *)
      MD593 AT %MD593 : UDINT := 16#00000000;  (* CDN[18].Tmax.(Ti |XYZ[0]): Темп. |Коорд.X *)
      MD594 AT %MD594 : UDINT := 16#00000000;  (* CDN[18].Tmax.(XYZ[1]|XYZ[2]): Коорд.Y|Коорд.Z *)
      MD595 AT %MD595 : UDINT := 16#00000000;  (* CDN[19].(ID|Tmid): Идент.|Tсред. *)
      MD596 AT %MD596 : UDINT := 16#00000000;  (* CDN[19].Tmin.(Ti |XYZ[0]): Темп. |Коорд.X *)
      MD597 AT %MD597 : UDINT := 16#00000000;  (* CDN[19].Tmin.(XYZ[1]|XYZ[2]): Коорд.Y|Коорд.Z *)
      MD598 AT %MD598 : UDINT := 16#00000000;  (* CDN[19].Tmax.(Ti |XYZ[0]): Темп. |Коорд.X *)
      MD599 AT %MD599 : UDINT := 16#00000000;  (* CDN[19].Tmax.(XYZ[1]|XYZ[2]): Коорд.Y|Коорд.Z *)
      MD600 AT %MD600 : UDINT := 16#00000000;  (* CDN[20].(ID|Tmid): Идент.|Tсред. *)
      MD601 AT %MD601 : UDINT := 16#00000000;  (* CDN[20].Tmin.(Ti |XYZ[0]): Темп. |Коорд.X *)
      MD602 AT %MD602 : UDINT := 16#00000000;  (* CDN[20].Tmin.(XYZ[1]|XYZ[2]): Коорд.Y|Коорд.Z *)
      MD603 AT %MD603 : UDINT := 16#00000000;  (* CDN[20].Tmax.(Ti |XYZ[0]): Темп. |Коорд.X *)
      MD604 AT %MD604 : UDINT := 16#00000000;  (* CDN[20].Tmax.(XYZ[1]|XYZ[2]): Коорд.Y|Коорд.Z *)
      MD605 AT %MD605 : UDINT := 16#00000000;  (* CDN[21].(ID|Tmid): Идент.|Tсред. *)
      MD606 AT %MD606 : UDINT := 16#00000000;  (* CDN[21].Tmin.(Ti |XYZ[0]): Темп. |Коорд.X *)
      MD607 AT %MD607 : UDINT := 16#00000000;  (* CDN[21].Tmin.(XYZ[1]|XYZ[2]): Коорд.Y|Коорд.Z *)
      MD608 AT %MD608 : UDINT := 16#00000000;  (* CDN[21].Tmax.(Ti |XYZ[0]): Темп. |Коорд.X *)
      MD609 AT %MD609 : UDINT := 16#00000000;  (* CDN[21].Tmax.(XYZ[1]|XYZ[2]): Коорд.Y|Коорд.Z *)
      MD610 AT %MD610 : UDINT := 16#00000000;  (* CDN[22].(ID|Tmid): Идент.|Tсред. *)
      MD611 AT %MD611 : UDINT := 16#00000000;  (* CDN[22].Tmin.(Ti |XYZ[0]): Темп. |Коорд.X *)
      MD612 AT %MD612 : UDINT := 16#00000000;  (* CDN[22].Tmin.(XYZ[1]|XYZ[2]): Коорд.Y|Коорд.Z *)
      MD613 AT %MD613 : UDINT := 16#00000000;  (* CDN[22].Tmax.(Ti |XYZ[0]): Темп. |Коорд.X *)
      MD614 AT %MD614 : UDINT := 16#00000000;  (* CDN[22].Tmax.(XYZ[1]|XYZ[2]): Коорд.Y|Коорд.Z *)
      MD615 AT %MD615 : UDINT := 16#00000000;  (* CDN[23].(ID|Tmid): Идент.|Tсред. *)
      MD616 AT %MD616 : UDINT := 16#00000000;  (* CDN[23].Tmin.(Ti |XYZ[0]): Темп. |Коорд.X *)
      MD617 AT %MD617 : UDINT := 16#00000000;  (* CDN[23].Tmin.(XYZ[1]|XYZ[2]): Коорд.Y|Коорд.Z *)
      MD618 AT %MD618 : UDINT := 16#00000000;  (* CDN[23].Tmax.(Ti |XYZ[0]): Темп. |Коорд.X *)
      MD619 AT %MD619 : UDINT := 16#00000000;  (* CDN[23].Tmax.(XYZ[1]|XYZ[2]): Коорд.Y|Коорд.Z *)
      MD620 AT %MD620 : UDINT := 16#00000000;  (* CDN[24].(ID|Tmid): Идент.|Tсред. *)
      MD621 AT %MD621 : UDINT := 16#00000000;  (* CDN[24].Tmin.(Ti |XYZ[0]): Темп. |Коорд.X *)
      MD622 AT %MD622 : UDINT := 16#00000000;  (* CDN[24].Tmin.(XYZ[1]|XYZ[2]): Коорд.Y|Коорд.Z *)
      MD623 AT %MD623 : UDINT := 16#00000000;  (* CDN[24].Tmax.(Ti |XYZ[0]): Темп. |Коорд.X *)
      MD624 AT %MD624 : UDINT := 16#00000000;  (* CDN[24].Tmax.(XYZ[1]|XYZ[2]): Коорд.Y|Коорд.Z *)
      MD625 AT %MD625 : UDINT := 16#00000000;  (* CDN[25].(ID|Tmid): Идент.|Tсред. *)
      MD626 AT %MD626 : UDINT := 16#00000000;  (* CDN[25].Tmin.(Ti |XYZ[0]): Темп. |Коорд.X *)
      MD627 AT %MD627 : UDINT := 16#00000000;  (* CDN[25].Tmin.(XYZ[1]|XYZ[2]): Коорд.Y|Коорд.Z *)
      MD628 AT %MD628 : UDINT := 16#00000000;  (* CDN[25].Tmax.(Ti |XYZ[0]): Темп. |Коорд.X *)
      MD629 AT %MD629 : UDINT := 16#00000000;  (* CDN[25].Tmax.(XYZ[1]|XYZ[2]): Коорд.Y|Коорд.Z *)
      MD630 AT %MD630 : UDINT := 16#00000000;  (* CDN[26].(ID|Tmid): Идент.|Tсред. *)
      MD631 AT %MD631 : UDINT := 16#00000000;  (* CDN[26].Tmin.(Ti |XYZ[0]): Темп. |Коорд.X *)
      MD632 AT %MD632 : UDINT := 16#00000000;  (* CDN[26].Tmin.(XYZ[1]|XYZ[2]): Коорд.Y|Коорд.Z *)
      MD633 AT %MD633 : UDINT := 16#00000000;  (* CDN[26].Tmax.(Ti |XYZ[0]): Темп. |Коорд.X *)
      MD634 AT %MD634 : UDINT := 16#00000000;  (* CDN[26].Tmax.(XYZ[1]|XYZ[2]): Коорд.Y|Коорд.Z *)
      MD635 AT %MD635 : UDINT := 16#00000000;  (* CDN[27].(ID|Tmid): Идент.|Tсред. *)
      MD636 AT %MD636 : UDINT := 16#00000000;  (* CDN[27].Tmin.(Ti |XYZ[0]): Темп. |Коорд.X *)
      MD637 AT %MD637 : UDINT := 16#00000000;  (* CDN[27].Tmin.(XYZ[1]|XYZ[2]): Коорд.Y|Коорд.Z *)
      MD638 AT %MD638 : UDINT := 16#00000000;  (* CDN[27].Tmax.(Ti |XYZ[0]): Темп. |Коорд.X *)
      MD639 AT %MD639 : UDINT := 16#00000000;  (* CDN[27].Tmax.(XYZ[1]|XYZ[2]): Коорд.Y|Коорд.Z *)
      MD640 AT %MD640 : UDINT := 16#00000000;  (* CDN[28].(ID|Tmid): Идент.|Tсред. *)
      MD641 AT %MD641 : UDINT := 16#00000000;  (* CDN[28].Tmin.(Ti |XYZ[0]): Темп. |Коорд.X *)
      MD642 AT %MD642 : UDINT := 16#00000000;  (* CDN[28].Tmin.(XYZ[1]|XYZ[2]): Коорд.Y|Коорд.Z *)
      MD643 AT %MD643 : UDINT := 16#00000000;  (* CDN[28].Tmax.(Ti |XYZ[0]): Темп. |Коорд.X *)
      MD644 AT %MD644 : UDINT := 16#00000000;  (* CDN[28].Tmax.(XYZ[1]|XYZ[2]): Коорд.Y|Коорд.Z *)
      MD645 AT %MD645 : UDINT := 16#00000000;  (* CDN[29].(ID|Tmid): Идент.|Tсред. *)
      MD646 AT %MD646 : UDINT := 16#00000000;  (* CDN[29].Tmin.(Ti |XYZ[0]): Темп. |Коорд.X *)
      MD647 AT %MD647 : UDINT := 16#00000000;  (* CDN[29].Tmin.(XYZ[1]|XYZ[2]): Коорд.Y|Коорд.Z *)
      MD648 AT %MD648 : UDINT := 16#00000000;  (* CDN[29].Tmax.(Ti |XYZ[0]): Темп. |Коорд.X *)
      MD649 AT %MD649 : UDINT := 16#00000000;  (* CDN[29].Tmax.(XYZ[1]|XYZ[2]): Коорд.Y|Коорд.Z *)
      MD650 AT %MD650 : UDINT := 16#00000000;  (* CDN[30].(ID|Tmid): Идент.|Tсред. *)
      MD651 AT %MD651 : UDINT := 16#00000000;  (* CDN[30].Tmin.(Ti |XYZ[0]): Темп. |Коорд.X *)
      MD652 AT %MD652 : UDINT := 16#00000000;  (* CDN[30].Tmin.(XYZ[1]|XYZ[2]): Коорд.Y|Коорд.Z *)
      MD653 AT %MD653 : UDINT := 16#00000000;  (* CDN[30].Tmax.(Ti |XYZ[0]): Темп. |Коорд.X *)
      MD654 AT %MD654 : UDINT := 16#00000000;  (* CDN[30].Tmax.(XYZ[1]|XYZ[2]): Коорд.Y|Коорд.Z *)
      MD655 AT %MD655 : UDINT := 16#00000000;  (* CDN[31].(ID|Tmid): Идент.|Tсред. *)
      MD656 AT %MD656 : UDINT := 16#00000000;  (* CDN[31].Tmin.(Ti |XYZ[0]): Темп. |Коорд.X *)
      MD657 AT %MD657 : UDINT := 16#00000000;  (* CDN[31].Tmin.(XYZ[1]|XYZ[2]): Коорд.Y|Коорд.Z *)
      MD658 AT %MD658 : UDINT := 16#00000000;  (* CDN[31].Tmax.(Ti |XYZ[0]): Темп. |Коорд.X *)
      MD659 AT %MD659 : UDINT := 16#00000000;  (* CDN[31].Tmax.(XYZ[1]|XYZ[2]): Коорд.Y|Коорд.Z *)
      MD660 AT %MD660 : UDINT := 16#00000000;  (* CDN[32].(ID|Tmid): Идент.|Tсред. *)
      MD661 AT %MD661 : UDINT := 16#00000000;  (* CDN[32].Tmin.(Ti |XYZ[0]): Темп. |Коорд.X *)
      MD662 AT %MD662 : UDINT := 16#00000000;  (* CDN[32].Tmin.(XYZ[1]|XYZ[2]): Коорд.Y|Коорд.Z *)
      MD663 AT %MD663 : UDINT := 16#00000000;  (* CDN[32].Tmax.(Ti |XYZ[0]): Темп. |Коорд.X *)
      MD664 AT %MD664 : UDINT := 16#00000000;  (* CDN[32].Tmax.(XYZ[1]|XYZ[2]): Коорд.Y|Коорд.Z *)
      MD665 AT %MD665 : UDINT := 16#00000000;  (* CDN[33].(ID|Tmid): Идент.|Tсред. *)
      MD666 AT %MD666 : UDINT := 16#00000000;  (* CDN[33].Tmin.(Ti |XYZ[0]): Темп. |Коорд.X *)
      MD667 AT %MD667 : UDINT := 16#00000000;  (* CDN[33].Tmin.(XYZ[1]|XYZ[2]): Коорд.Y|Коорд.Z *)
      MD668 AT %MD668 : UDINT := 16#00000000;  (* CDN[33].Tmax.(Ti |XYZ[0]): Темп. |Коорд.X *)
      MD669 AT %MD669 : UDINT := 16#00000000;  (* CDN[33].Tmax.(XYZ[1]|XYZ[2]): Коорд.Y|Коорд.Z *)
      MD670 AT %MD670 : UDINT := 16#00000000;  (* CDN[34].(ID|Tmid): Идент.|Tсред. *)
      MD671 AT %MD671 : UDINT := 16#00000000;  (* CDN[34].Tmin.(Ti |XYZ[0]): Темп. |Коорд.X *)
      MD672 AT %MD672 : UDINT := 16#00000000;  (* CDN[34].Tmin.(XYZ[1]|XYZ[2]): Коорд.Y|Коорд.Z *)
      MD673 AT %MD673 : UDINT := 16#00000000;  (* CDN[34].Tmax.(Ti |XYZ[0]): Темп. |Коорд.X *)
      MD674 AT %MD674 : UDINT := 16#00000000;  (* CDN[34].Tmax.(XYZ[1]|XYZ[2]): Коорд.Y|Коорд.Z *)
      MD675 AT %MD675 : UDINT := 16#00000000;  (* CDN[35].(ID|Tmid): Идент.|Tсред. *)
      MD676 AT %MD676 : UDINT := 16#00000000;  (* CDN[35].Tmin.(Ti |XYZ[0]): Темп. |Коорд.X *)
      MD677 AT %MD677 : UDINT := 16#00000000;  (* CDN[35].Tmin.(XYZ[1]|XYZ[2]): Коорд.Y|Коорд.Z *)
      MD678 AT %MD678 : UDINT := 16#00000000;  (* CDN[35].Tmax.(Ti |XYZ[0]): Темп. |Коорд.X *)
      MD679 AT %MD679 : UDINT := 16#00000000;  (* CDN[35].Tmax.(XYZ[1]|XYZ[2]): Коорд.Y|Коорд.Z *)
      MD680 AT %MD680 : UDINT := 16#00000000;  (* CDN[36].(ID|Tmid): Идент.|Tсред. *)
      MD681 AT %MD681 : UDINT := 16#00000000;  (* CDN[36].Tmin.(Ti |XYZ[0]): Темп. |Коорд.X *)
      MD682 AT %MD682 : UDINT := 16#00000000;  (* CDN[36].Tmin.(XYZ[1]|XYZ[2]): Коорд.Y|Коорд.Z *)
      MD683 AT %MD683 : UDINT := 16#00000000;  (* CDN[36].Tmax.(Ti |XYZ[0]): Темп. |Коорд.X *)
      MD684 AT %MD684 : UDINT := 16#00000000;  (* CDN[36].Tmax.(XYZ[1]|XYZ[2]): Коорд.Y|Коорд.Z *)
      MD685 AT %MD685 : UDINT := 16#00000000;  (* CDN[37].(ID|Tmid): Идент.|Tсред. *)
      MD686 AT %MD686 : UDINT := 16#00000000;  (* CDN[37].Tmin.(Ti |XYZ[0]): Темп. |Коорд.X *)
      MD687 AT %MD687 : UDINT := 16#00000000;  (* CDN[37].Tmin.(XYZ[1]|XYZ[2]): Коорд.Y|Коорд.Z *)
      MD688 AT %MD688 : UDINT := 16#00000000;  (* CDN[37].Tmax.(Ti |XYZ[0]): Темп. |Коорд.X *)
      MD689 AT %MD689 : UDINT := 16#00000000;  (* CDN[37].Tmax.(XYZ[1]|XYZ[2]): Коорд.Y|Коорд.Z *)
      MD690 AT %MD690 : UDINT := 16#00000000;  (* CDN[38].(ID|Tmid): Идент.|Tсред. *)
      MD691 AT %MD691 : UDINT := 16#00000000;  (* CDN[38].Tmin.(Ti |XYZ[0]): Темп. |Коорд.X *)
      MD692 AT %MD692 : UDINT := 16#00000000;  (* CDN[38].Tmin.(XYZ[1]|XYZ[2]): Коорд.Y|Коорд.Z *)
      MD693 AT %MD693 : UDINT := 16#00000000;  (* CDN[38].Tmax.(Ti |XYZ[0]): Темп. |Коорд.X *)
      MD694 AT %MD694 : UDINT := 16#00000000;  (* CDN[38].Tmax.(XYZ[1]|XYZ[2]): Коорд.Y|Коорд.Z *)
      MD695 AT %MD695 : UDINT := 16#00000000;  (* CDN[39].(ID|Tmid): Идент.|Tсред. *)
      MD696 AT %MD696 : UDINT := 16#00000000;  (* CDN[39].Tmin.(Ti |XYZ[0]): Темп. |Коорд.X *)
      MD697 AT %MD697 : UDINT := 16#00000000;  (* CDN[39].Tmin.(XYZ[1]|XYZ[2]): Коорд.Y|Коорд.Z *)
      MD698 AT %MD698 : UDINT := 16#00000000;  (* CDN[39].Tmax.(Ti |XYZ[0]): Темп. |Коорд.X *)
      MD699 AT %MD699 : UDINT := 16#00000000;  (* CDN[39].Tmax.(XYZ[1]|XYZ[2]): Коорд.Y|Коорд.Z *)
      MD700 AT %MD700 : UDINT := 16#00000000;  (* CDN[40].(ID|Tmid): Идент.|Tсред. *)
      MD701 AT %MD701 : UDINT := 16#00000000;  (* CDN[40].Tmin.(Ti |XYZ[0]): Темп. |Коорд.X *)
      MD702 AT %MD702 : UDINT := 16#00000000;  (* CDN[40].Tmin.(XYZ[1]|XYZ[2]): Коорд.Y|Коорд.Z *)
      MD703 AT %MD703 : UDINT := 16#00000000;  (* CDN[40].Tmax.(Ti |XYZ[0]): Темп. |Коорд.X *)
      MD704 AT %MD704 : UDINT := 16#00000000;  (* CDN[40].Tmax.(XYZ[1]|XYZ[2]): Коорд.Y|Коорд.Z *)
      MD705 AT %MD705 : UDINT := 16#00000000;  (* CDN[41].(ID|Tmid): Идент.|Tсред. *)
      MD706 AT %MD706 : UDINT := 16#00000000;  (* CDN[41].Tmin.(Ti |XYZ[0]): Темп. |Коорд.X *)
      MD707 AT %MD707 : UDINT := 16#00000000;  (* CDN[41].Tmin.(XYZ[1]|XYZ[2]): Коорд.Y|Коорд.Z *)
      MD708 AT %MD708 : UDINT := 16#00000000;  (* CDN[41].Tmax.(Ti |XYZ[0]): Темп. |Коорд.X *)
      MD709 AT %MD709 : UDINT := 16#00000000;  (* CDN[41].Tmax.(XYZ[1]|XYZ[2]): Коорд.Y|Коорд.Z *)
      MD710 AT %MD710 : UDINT := 16#00000000;  (* CDN[42].(ID|Tmid): Идент.|Tсред. *)
      MD711 AT %MD711 : UDINT := 16#00000000;  (* CDN[42].Tmin.(Ti |XYZ[0]): Темп. |Коорд.X *)
      MD712 AT %MD712 : UDINT := 16#00000000;  (* CDN[42].Tmin.(XYZ[1]|XYZ[2]): Коорд.Y|Коорд.Z *)
      MD713 AT %MD713 : UDINT := 16#00000000;  (* CDN[42].Tmax.(Ti |XYZ[0]): Темп. |Коорд.X *)
      MD714 AT %MD714 : UDINT := 16#00000000;  (* CDN[42].Tmax.(XYZ[1]|XYZ[2]): Коорд.Y|Коорд.Z *)
      MD715 AT %MD715 : UDINT := 16#00000000;  (* CDN[43].(ID|Tmid): Идент.|Tсред. *)
      MD716 AT %MD716 : UDINT := 16#00000000;  (* CDN[43].Tmin.(Ti |XYZ[0]): Темп. |Коорд.X *)
      MD717 AT %MD717 : UDINT := 16#00000000;  (* CDN[43].Tmin.(XYZ[1]|XYZ[2]): Коорд.Y|Коорд.Z *)
      MD718 AT %MD718 : UDINT := 16#00000000;  (* CDN[43].Tmax.(Ti |XYZ[0]): Темп. |Коорд.X *)
      MD719 AT %MD719 : UDINT := 16#00000000;  (* CDN[43].Tmax.(XYZ[1]|XYZ[2]): Коорд.Y|Коорд.Z *)
      MD720 AT %MD720 : UDINT := 16#00000000;  (* CDN[44].(ID|Tmid): Идент.|Tсред. *)
      MD721 AT %MD721 : UDINT := 16#00000000;  (* CDN[44].Tmin.(Ti |XYZ[0]): Темп. |Коорд.X *)
      MD722 AT %MD722 : UDINT := 16#00000000;  (* CDN[44].Tmin.(XYZ[1]|XYZ[2]): Коорд.Y|Коорд.Z *)
      MD723 AT %MD723 : UDINT := 16#00000000;  (* CDN[44].Tmax.(Ti |XYZ[0]): Темп. |Коорд.X *)
      MD724 AT %MD724 : UDINT := 16#00000000;  (* CDN[44].Tmax.(XYZ[1]|XYZ[2]): Коорд.Y|Коорд.Z *)
      MD725 AT %MD725 : UDINT := 16#00000000;  (* CDN[45].(ID|Tmid): Идент.|Tсред. *)
      MD726 AT %MD726 : UDINT := 16#00000000;  (* CDN[45].Tmin.(Ti |XYZ[0]): Темп. |Коорд.X *)
      MD727 AT %MD727 : UDINT := 16#00000000;  (* CDN[45].Tmin.(XYZ[1]|XYZ[2]): Коорд.Y|Коорд.Z *)
      MD728 AT %MD728 : UDINT := 16#00000000;  (* CDN[45].Tmax.(Ti |XYZ[0]): Темп. |Коорд.X *)
      MD729 AT %MD729 : UDINT := 16#00000000;  (* CDN[45].Tmax.(XYZ[1]|XYZ[2]): Коорд.Y|Коорд.Z *)
      MD730 AT %MD730 : UDINT := 16#00000000;  (* CDN[46].(ID|Tmid): Идент.|Tсред. *)
      MD731 AT %MD731 : UDINT := 16#00000000;  (* CDN[46].Tmin.(Ti |XYZ[0]): Темп. |Коорд.X *)
      MD732 AT %MD732 : UDINT := 16#00000000;  (* CDN[46].Tmin.(XYZ[1]|XYZ[2]): Коорд.Y|Коорд.Z *)
      MD733 AT %MD733 : UDINT := 16#00000000;  (* CDN[46].Tmax.(Ti |XYZ[0]): Темп. |Коорд.X *)
      MD734 AT %MD734 : UDINT := 16#00000000;  (* CDN[46].Tmax.(XYZ[1]|XYZ[2]): Коорд.Y|Коорд.Z *)
      MD735 AT %MD735 : UDINT := 16#00000000;  (* CDN[47].(ID|Tmid): Идент.|Tсред. *)
      MD736 AT %MD736 : UDINT := 16#00000000;  (* CDN[47].Tmin.(Ti |XYZ[0]): Темп. |Коорд.X *)
      MD737 AT %MD737 : UDINT := 16#00000000;  (* CDN[47].Tmin.(XYZ[1]|XYZ[2]): Коорд.Y|Коорд.Z *)
      MD738 AT %MD738 : UDINT := 16#00000000;  (* CDN[47].Tmax.(Ti |XYZ[0]): Темп. |Коорд.X *)
      MD739 AT %MD739 : UDINT := 16#00000000;  (* CDN[47].Tmax.(XYZ[1]|XYZ[2]): Коорд.Y|Коорд.Z *)
      MD740 AT %MD740 : UDINT := 16#00000000;  (* CDN[48].(ID|Tmid): Идент.|Tсред. *)
      MD741 AT %MD741 : UDINT := 16#00000000;  (* CDN[48].Tmin.(Ti |XYZ[0]): Темп. |Коорд.X *)
      MD742 AT %MD742 : UDINT := 16#00000000;  (* CDN[48].Tmin.(XYZ[1]|XYZ[2]): Коорд.Y|Коорд.Z *)
      MD743 AT %MD743 : UDINT := 16#00000000;  (* CDN[48].Tmax.(Ti |XYZ[0]): Темп. |Коорд.X *)
      MD744 AT %MD744 : UDINT := 16#00000000;  (* CDN[48].Tmax.(XYZ[1]|XYZ[2]): Коорд.Y|Коорд.Z *)
      MD745 AT %MD745 : UDINT := 16#00000000;  (* CDN[49].(ID|Tmid): Идент.|Tсред. *)
      MD746 AT %MD746 : UDINT := 16#00000000;  (* CDN[49].Tmin.(Ti |XYZ[0]): Темп. |Коорд.X *)
      MD747 AT %MD747 : UDINT := 16#00000000;  (* CDN[49].Tmin.(XYZ[1]|XYZ[2]): Коорд.Y|Коорд.Z *)
      MD748 AT %MD748 : UDINT := 16#00000000;  (* CDN[49].Tmax.(Ti |XYZ[0]): Темп. |Коорд.X *)
      MD749 AT %MD749 : UDINT := 16#00000000;  (* CDN[49].Tmax.(XYZ[1]|XYZ[2]): Коорд.Y|Коорд.Z *)
      MD750 AT %MD750 : UDINT := 16#00000000;  (* CDN[50].(ID|Tmid): Идент.|Tсред. *)
      MD751 AT %MD751 : UDINT := 16#00000000;  (* CDN[50].Tmin.(Ti |XYZ[0]): Темп. |Коорд.X *)
      MD752 AT %MD752 : UDINT := 16#00000000;  (* CDN[50].Tmin.(XYZ[1]|XYZ[2]): Коорд.Y|Коорд.Z *)
      MD753 AT %MD753 : UDINT := 16#00000000;  (* CDN[50].Tmax.(Ti |XYZ[0]): Темп. |Коорд.X *)
      MD754 AT %MD754 : UDINT := 16#00000000;  (* CDN[50].Tmax.(XYZ[1]|XYZ[2]): Коорд.Y|Коорд.Z *)
      MD755 AT %MD755 : UDINT := 16#00000000;  (* CDN[51].(ID|Tmid): Идент.|Tсред. *)
      MD756 AT %MD756 : UDINT := 16#00000000;  (* CDN[51].Tmin.(Ti |XYZ[0]): Темп. |Коорд.X *)
      MD757 AT %MD757 : UDINT := 16#00000000;  (* CDN[51].Tmin.(XYZ[1]|XYZ[2]): Коорд.Y|Коорд.Z *)
      MD758 AT %MD758 : UDINT := 16#00000000;  (* CDN[51].Tmax.(Ti |XYZ[0]): Темп. |Коорд.X *)
      MD759 AT %MD759 : UDINT := 16#00000000;  (* CDN[51].Tmax.(XYZ[1]|XYZ[2]): Коорд.Y|Коорд.Z *)
      MD760 AT %MD760 : UDINT := 16#00000000;  (* CDN[52].(ID|Tmid): Идент.|Tсред. *)
      MD761 AT %MD761 : UDINT := 16#00000000;  (* CDN[52].Tmin.(Ti |XYZ[0]): Темп. |Коорд.X *)
      MD762 AT %MD762 : UDINT := 16#00000000;  (* CDN[52].Tmin.(XYZ[1]|XYZ[2]): Коорд.Y|Коорд.Z *)
      MD763 AT %MD763 : UDINT := 16#00000000;  (* CDN[52].Tmax.(Ti |XYZ[0]): Темп. |Коорд.X *)
      MD764 AT %MD764 : UDINT := 16#00000000;  (* CDN[52].Tmax.(XYZ[1]|XYZ[2]): Коорд.Y|Коорд.Z *)
      MD765 AT %MD765 : UDINT := 16#00000000;  (* CDN[53].(ID|Tmid): Идент.|Tсред. *)
      MD766 AT %MD766 : UDINT := 16#00000000;  (* CDN[53].Tmin.(Ti |XYZ[0]): Темп. |Коорд.X *)
      MD767 AT %MD767 : UDINT := 16#00000000;  (* CDN[53].Tmin.(XYZ[1]|XYZ[2]): Коорд.Y|Коорд.Z *)
      MD768 AT %MD768 : UDINT := 16#00000000;  (* CDN[53].Tmax.(Ti |XYZ[0]): Темп. |Коорд.X *)
      MD769 AT %MD769 : UDINT := 16#00000000;  (* CDN[53].Tmax.(XYZ[1]|XYZ[2]): Коорд.Y|Коорд.Z *)
      MD770 AT %MD770 : UDINT := 16#00000000;  (* CDN[54].(ID|Tmid): Идент.|Tсред. *)
      MD771 AT %MD771 : UDINT := 16#00000000;  (* CDN[54].Tmin.(Ti |XYZ[0]): Темп. |Коорд.X *)
      MD772 AT %MD772 : UDINT := 16#00000000;  (* CDN[54].Tmin.(XYZ[1]|XYZ[2]): Коорд.Y|Коорд.Z *)
      MD773 AT %MD773 : UDINT := 16#00000000;  (* CDN[54].Tmax.(Ti |XYZ[0]): Темп. |Коорд.X *)
      MD774 AT %MD774 : UDINT := 16#00000000;  (* CDN[54].Tmax.(XYZ[1]|XYZ[2]): Коорд.Y|Коорд.Z *)
      MD775 AT %MD775 : UDINT := 16#00000000;  (* CDN[55].(ID|Tmid): Идент.|Tсред. *)
      MD776 AT %MD776 : UDINT := 16#00000000;  (* CDN[55].Tmin.(Ti |XYZ[0]): Темп. |Коорд.X *)
      MD777 AT %MD777 : UDINT := 16#00000000;  (* CDN[55].Tmin.(XYZ[1]|XYZ[2]): Коорд.Y|Коорд.Z *)
      MD778 AT %MD778 : UDINT := 16#00000000;  (* CDN[55].Tmax.(Ti |XYZ[0]): Темп. |Коорд.X *)
      MD779 AT %MD779 : UDINT := 16#00000000;  (* CDN[55].Tmax.(XYZ[1]|XYZ[2]): Коорд.Y|Коорд.Z *)
      MD780 AT %MD780 : UDINT := 16#00000000;  (* CDN[56].(ID|Tmid): Идент.|Tсред. *)
      MD781 AT %MD781 : UDINT := 16#00000000;  (* CDN[56].Tmin.(Ti |XYZ[0]): Темп. |Коорд.X *)
      MD782 AT %MD782 : UDINT := 16#00000000;  (* CDN[56].Tmin.(XYZ[1]|XYZ[2]): Коорд.Y|Коорд.Z *)
      MD783 AT %MD783 : UDINT := 16#00000000;  (* CDN[56].Tmax.(Ti |XYZ[0]): Темп. |Коорд.X *)
      MD784 AT %MD784 : UDINT := 16#00000000;  (* CDN[56].Tmax.(XYZ[1]|XYZ[2]): Коорд.Y|Коорд.Z *)
      MD785 AT %MD785 : UDINT := 16#00000000;  (* CDN[57].(ID|Tmid): Идент.|Tсред. *)
      MD786 AT %MD786 : UDINT := 16#00000000;  (* CDN[57].Tmin.(Ti |XYZ[0]): Темп. |Коорд.X *)
      MD787 AT %MD787 : UDINT := 16#00000000;  (* CDN[57].Tmin.(XYZ[1]|XYZ[2]): Коорд.Y|Коорд.Z *)
      MD788 AT %MD788 : UDINT := 16#00000000;  (* CDN[57].Tmax.(Ti |XYZ[0]): Темп. |Коорд.X *)
      MD789 AT %MD789 : UDINT := 16#00000000;  (* CDN[57].Tmax.(XYZ[1]|XYZ[2]): Коорд.Y|Коорд.Z *)
      MD790 AT %MD790 : UDINT := 16#00000000;  (* CDN[58].(ID|Tmid): Идент.|Tсред. *)
      MD791 AT %MD791 : UDINT := 16#00000000;  (* CDN[58].Tmin.(Ti |XYZ[0]): Темп. |Коорд.X *)
      MD792 AT %MD792 : UDINT := 16#00000000;  (* CDN[58].Tmin.(XYZ[1]|XYZ[2]): Коорд.Y|Коорд.Z *)
      MD793 AT %MD793 : UDINT := 16#00000000;  (* CDN[58].Tmax.(Ti |XYZ[0]): Темп. |Коорд.X *)
      MD794 AT %MD794 : UDINT := 16#00000000;  (* CDN[58].Tmax.(XYZ[1]|XYZ[2]): Коорд.Y|Коорд.Z *)
      MD795 AT %MD795 : UDINT := 16#00000000;  (* CDN[59].(ID|Tmid): Идент.|Tсред. *)
      MD796 AT %MD796 : UDINT := 16#00000000;  (* CDN[59].Tmin.(Ti |XYZ[0]): Темп. |Коорд.X *)
      MD797 AT %MD797 : UDINT := 16#00000000;  (* CDN[59].Tmin.(XYZ[1]|XYZ[2]): Коорд.Y|Коорд.Z *)
      MD798 AT %MD798 : UDINT := 16#00000000;  (* CDN[59].Tmax.(Ti |XYZ[0]): Темп. |Коорд.X *)
      MD799 AT %MD799 : UDINT := 16#00000000;  (* CDN[59].Tmax.(XYZ[1]|XYZ[2]): Коорд.Y|Коорд.Z *)
      MD800 AT %MD800 : UDINT := 16#00000000;  (* CDN[60].(ID|Tmid): Идент.|Tсред. *)
      MD801 AT %MD801 : UDINT := 16#00000000;  (* CDN[60].Tmin.(Ti |XYZ[0]): Темп. |Коорд.X *)
      MD802 AT %MD802 : UDINT := 16#00000000;  (* CDN[60].Tmin.(XYZ[1]|XYZ[2]): Коорд.Y|Коорд.Z *)
      MD803 AT %MD803 : UDINT := 16#00000000;  (* CDN[60].Tmax.(Ti |XYZ[0]): Темп. |Коорд.X *)
      MD804 AT %MD804 : UDINT := 16#00000000;  (* CDN[60].Tmax.(XYZ[1]|XYZ[2]): Коорд.Y|Коорд.Z *)
      MD805 AT %MD805 : UDINT := 16#00000000;  (* CDN[61].(ID|Tmid): Идент.|Tсред. *)
      MD806 AT %MD806 : UDINT := 16#00000000;  (* CDN[61].Tmin.(Ti |XYZ[0]): Темп. |Коорд.X *)
      MD807 AT %MD807 : UDINT := 16#00000000;  (* CDN[61].Tmin.(XYZ[1]|XYZ[2]): Коорд.Y|Коорд.Z *)
      MD808 AT %MD808 : UDINT := 16#00000000;  (* CDN[61].Tmax.(Ti |XYZ[0]): Темп. |Коорд.X *)
      MD809 AT %MD809 : UDINT := 16#00000000;  (* CDN[61].Tmax.(XYZ[1]|XYZ[2]): Коорд.Y|Коорд.Z *)
      MD810 AT %MD810 : UDINT := 16#00000000;  (* CDN[62].(ID|Tmid): Идент.|Tсред. *)
      MD811 AT %MD811 : UDINT := 16#00000000;  (* CDN[62].Tmin.(Ti |XYZ[0]): Темп. |Коорд.X *)
      MD812 AT %MD812 : UDINT := 16#00000000;  (* CDN[62].Tmin.(XYZ[1]|XYZ[2]): Коорд.Y|Коорд.Z *)
      MD813 AT %MD813 : UDINT := 16#00000000;  (* CDN[62].Tmax.(Ti |XYZ[0]): Темп. |Коорд.X *)
      MD814 AT %MD814 : UDINT := 16#00000000;  (* CDN[62].Tmax.(XYZ[1]|XYZ[2]): Коорд.Y|Коорд.Z *)
      MD815 AT %MD815 : UDINT := 16#00000000;  (* CDN[63].(ID|Tmid): Идент.|Tсред. *)
      MD816 AT %MD816 : UDINT := 16#00000000;  (* CDN[63].Tmin.(Ti |XYZ[0]): Темп. |Коорд.X *)
      MD817 AT %MD817 : UDINT := 16#00000000;  (* CDN[63].Tmin.(XYZ[1]|XYZ[2]): Коорд.Y|Коорд.Z *)
      MD818 AT %MD818 : UDINT := 16#00000000;  (* CDN[63].Tmax.(Ti |XYZ[0]): Темп. |Коорд.X *)
      MD819 AT %MD819 : UDINT := 16#00000000;  (* CDN[63].Tmax.(XYZ[1]|XYZ[2]): Коорд.Y|Коорд.Z *)
      MD820 AT %MD820 : UDINT := 16#00000000;  (* CDN[64].(ID|Tmid): Идент.|Tсред. *)
      MD821 AT %MD821 : UDINT := 16#00000000;  (* CDN[64].Tmin.(Ti |XYZ[0]): Темп. |Коорд.X *)
      MD822 AT %MD822 : UDINT := 16#00000000;  (* CDN[64].Tmin.(XYZ[1]|XYZ[2]): Коорд.Y|Коорд.Z *)
      MD823 AT %MD823 : UDINT := 16#00000000;  (* CDN[64].Tmax.(Ti |XYZ[0]): Темп. |Коорд.X *)
      MD824 AT %MD824 : UDINT := 16#00000000;  (* CDN[64].Tmax.(XYZ[1]|XYZ[2]): Коорд.Y|Коорд.Z *)
      MD825 AT %MD825 : UDINT := 16#00000000;  (* CDN[65].(ID|Tmid): Идент.|Tсред. *)
      MD826 AT %MD826 : UDINT := 16#00000000;  (* CDN[65].Tmin.(Ti |XYZ[0]): Темп. |Коорд.X *)
      MD827 AT %MD827 : UDINT := 16#00000000;  (* CDN[65].Tmin.(XYZ[1]|XYZ[2]): Коорд.Y|Коорд.Z *)
      MD828 AT %MD828 : UDINT := 16#00000000;  (* CDN[65].Tmax.(Ti |XYZ[0]): Темп. |Коорд.X *)
      MD829 AT %MD829 : UDINT := 16#00000000;  (* CDN[65].Tmax.(XYZ[1]|XYZ[2]): Коорд.Y|Коорд.Z *)
      MD830 AT %MD830 : UDINT := 16#00000000;  (* CDN[66].(ID|Tmid): Идент.|Tсред. *)
      MD831 AT %MD831 : UDINT := 16#00000000;  (* CDN[66].Tmin.(Ti |XYZ[0]): Темп. |Коорд.X *)
      MD832 AT %MD832 : UDINT := 16#00000000;  (* CDN[66].Tmin.(XYZ[1]|XYZ[2]): Коорд.Y|Коорд.Z *)
      MD833 AT %MD833 : UDINT := 16#00000000;  (* CDN[66].Tmax.(Ti |XYZ[0]): Темп. |Коорд.X *)
      MD834 AT %MD834 : UDINT := 16#00000000;  (* CDN[66].Tmax.(XYZ[1]|XYZ[2]): Коорд.Y|Коорд.Z *)
      MD835 AT %MD835 : UDINT := 16#00000000;  (* CDN[67].(ID|Tmid): Идент.|Tсред. *)
      MD836 AT %MD836 : UDINT := 16#00000000;  (* CDN[67].Tmin.(Ti |XYZ[0]): Темп. |Коорд.X *)
      MD837 AT %MD837 : UDINT := 16#00000000;  (* CDN[67].Tmin.(XYZ[1]|XYZ[2]): Коорд.Y|Коорд.Z *)
      MD838 AT %MD838 : UDINT := 16#00000000;  (* CDN[67].Tmax.(Ti |XYZ[0]): Темп. |Коорд.X *)
      MD839 AT %MD839 : UDINT := 16#00000000;  (* CDN[67].Tmax.(XYZ[1]|XYZ[2]): Коорд.Y|Коорд.Z *)
      MD840 AT %MD840 : UDINT := 16#00000000;  (* CDN[68].(ID|Tmid): Идент.|Tсред. *)
      MD841 AT %MD841 : UDINT := 16#00000000;  (* CDN[68].Tmin.(Ti |XYZ[0]): Темп. |Коорд.X *)
      MD842 AT %MD842 : UDINT := 16#00000000;  (* CDN[68].Tmin.(XYZ[1]|XYZ[2]): Коорд.Y|Коорд.Z *)
      MD843 AT %MD843 : UDINT := 16#00000000;  (* CDN[68].Tmax.(Ti |XYZ[0]): Темп. |Коорд.X *)
      MD844 AT %MD844 : UDINT := 16#00000000;  (* CDN[68].Tmax.(XYZ[1]|XYZ[2]): Коорд.Y|Коорд.Z *)
      MD845 AT %MD845 : UDINT := 16#00000000;  (* CDN[69].(ID|Tmid): Идент.|Tсред. *)
      MD846 AT %MD846 : UDINT := 16#00000000;  (* CDN[69].Tmin.(Ti |XYZ[0]): Темп. |Коорд.X *)
      MD847 AT %MD847 : UDINT := 16#00000000;  (* CDN[69].Tmin.(XYZ[1]|XYZ[2]): Коорд.Y|Коорд.Z *)
      MD848 AT %MD848 : UDINT := 16#00000000;  (* CDN[69].Tmax.(Ti |XYZ[0]): Темп. |Коорд.X *)
      MD849 AT %MD849 : UDINT := 16#00000000;  (* CDN[69].Tmax.(XYZ[1]|XYZ[2]): Коорд.Y|Коорд.Z *)
      MD850 AT %MD850 : UDINT := 16#00000000;  (* CDN[70].(ID|Tmid): Идент.|Tсред. *)
      MD851 AT %MD851 : UDINT := 16#00000000;  (* CDN[70].Tmin.(Ti |XYZ[0]): Темп. |Коорд.X *)
      MD852 AT %MD852 : UDINT := 16#00000000;  (* CDN[70].Tmin.(XYZ[1]|XYZ[2]): Коорд.Y|Коорд.Z *)
      MD853 AT %MD853 : UDINT := 16#00000000;  (* CDN[70].Tmax.(Ti |XYZ[0]): Темп. |Коорд.X *)
      MD854 AT %MD854 : UDINT := 16#00000000;  (* CDN[70].Tmax.(XYZ[1]|XYZ[2]): Коорд.Y|Коорд.Z *)
      MD855 AT %MD855 : UDINT := 16#00000000;  (* CDN[71].(ID|Tmid): Идент.|Tсред. *)
      MD856 AT %MD856 : UDINT := 16#00000000;  (* CDN[71].Tmin.(Ti |XYZ[0]): Темп. |Коорд.X *)
      MD857 AT %MD857 : UDINT := 16#00000000;  (* CDN[71].Tmin.(XYZ[1]|XYZ[2]): Коорд.Y|Коорд.Z *)
      MD858 AT %MD858 : UDINT := 16#00000000;  (* CDN[71].Tmax.(Ti |XYZ[0]): Темп. |Коорд.X *)
      MD859 AT %MD859 : UDINT := 16#00000000;  (* CDN[71].Tmax.(XYZ[1]|XYZ[2]): Коорд.Y|Коорд.Z *)
      MD860 AT %MD860 : UDINT := 16#00000000;  (* CDN[72].(ID|Tmid): Идент.|Tсред. *)
      MD861 AT %MD861 : UDINT := 16#00000000;  (* CDN[72].Tmin.(Ti |XYZ[0]): Темп. |Коорд.X *)
      MD862 AT %MD862 : UDINT := 16#00000000;  (* CDN[72].Tmin.(XYZ[1]|XYZ[2]): Коорд.Y|Коорд.Z *)
      MD863 AT %MD863 : UDINT := 16#00000000;  (* CDN[72].Tmax.(Ti |XYZ[0]): Темп. |Коорд.X *)
      MD864 AT %MD864 : UDINT := 16#00000000;  (* CDN[72].Tmax.(XYZ[1]|XYZ[2]): Коорд.Y|Коорд.Z *)
      MD865 AT %MD865 : UDINT := 16#00000000;  (* CDN[73].(ID|Tmid): Идент.|Tсред. *)
      MD866 AT %MD866 : UDINT := 16#00000000;  (* CDN[73].Tmin.(Ti |XYZ[0]): Темп. |Коорд.X *)
      MD867 AT %MD867 : UDINT := 16#00000000;  (* CDN[73].Tmin.(XYZ[1]|XYZ[2]): Коорд.Y|Коорд.Z *)
      MD868 AT %MD868 : UDINT := 16#00000000;  (* CDN[73].Tmax.(Ti |XYZ[0]): Темп. |Коорд.X *)
      MD869 AT %MD869 : UDINT := 16#00000000;  (* CDN[73].Tmax.(XYZ[1]|XYZ[2]): Коорд.Y|Коорд.Z *)
      MD870 AT %MD870 : UDINT := 16#00000000;  (* CDN[74].(ID|Tmid): Идент.|Tсред. *)
      MD871 AT %MD871 : UDINT := 16#00000000;  (* CDN[74].Tmin.(Ti |XYZ[0]): Темп. |Коорд.X *)
      MD872 AT %MD872 : UDINT := 16#00000000;  (* CDN[74].Tmin.(XYZ[1]|XYZ[2]): Коорд.Y|Коорд.Z *)
      MD873 AT %MD873 : UDINT := 16#00000000;  (* CDN[74].Tmax.(Ti |XYZ[0]): Темп. |Коорд.X *)
      MD874 AT %MD874 : UDINT := 16#00000000;  (* CDN[74].Tmax.(XYZ[1]|XYZ[2]): Коорд.Y|Коорд.Z *)
      MD875 AT %MD875 : UDINT := 16#00000000;  (* CDN[75].(ID|Tmid): Идент.|Tсред. *)
      MD876 AT %MD876 : UDINT := 16#00000000;  (* CDN[75].Tmin.(Ti |XYZ[0]): Темп. |Коорд.X *)
      MD877 AT %MD877 : UDINT := 16#00000000;  (* CDN[75].Tmin.(XYZ[1]|XYZ[2]): Коорд.Y|Коорд.Z *)
      MD878 AT %MD878 : UDINT := 16#00000000;  (* CDN[75].Tmax.(Ti |XYZ[0]): Темп. |Коорд.X *)
      MD879 AT %MD879 : UDINT := 16#00000000;  (* CDN[75].Tmax.(XYZ[1]|XYZ[2]): Коорд.Y|Коорд.Z *)
      MD880 AT %MD880 : UDINT := 16#00000000;  (* CDN[76].(ID|Tmid): Идент.|Tсред. *)
      MD881 AT %MD881 : UDINT := 16#00000000;  (* CDN[76].Tmin.(Ti |XYZ[0]): Темп. |Коорд.X *)
      MD882 AT %MD882 : UDINT := 16#00000000;  (* CDN[76].Tmin.(XYZ[1]|XYZ[2]): Коорд.Y|Коорд.Z *)
      MD883 AT %MD883 : UDINT := 16#00000000;  (* CDN[76].Tmax.(Ti |XYZ[0]): Темп. |Коорд.X *)
      MD884 AT %MD884 : UDINT := 16#00000000;  (* CDN[76].Tmax.(XYZ[1]|XYZ[2]): Коорд.Y|Коорд.Z *)
      MD885 AT %MD885 : UDINT := 16#00000000;  (* CDN[77].(ID|Tmid): Идент.|Tсред. *)
      MD886 AT %MD886 : UDINT := 16#00000000;  (* CDN[77].Tmin.(Ti |XYZ[0]): Темп. |Коорд.X *)
      MD887 AT %MD887 : UDINT := 16#00000000;  (* CDN[77].Tmin.(XYZ[1]|XYZ[2]): Коорд.Y|Коорд.Z *)
      MD888 AT %MD888 : UDINT := 16#00000000;  (* CDN[77].Tmax.(Ti |XYZ[0]): Темп. |Коорд.X *)
      MD889 AT %MD889 : UDINT := 16#00000000;  (* CDN[77].Tmax.(XYZ[1]|XYZ[2]): Коорд.Y|Коорд.Z *)
      MD890 AT %MD890 : UDINT := 16#00000000;  (* CDN[78].(ID|Tmid): Идент.|Tсред. *)
      MD891 AT %MD891 : UDINT := 16#00000000;  (* CDN[78].Tmin.(Ti |XYZ[0]): Темп. |Коорд.X *)
      MD892 AT %MD892 : UDINT := 16#00000000;  (* CDN[78].Tmin.(XYZ[1]|XYZ[2]): Коорд.Y|Коорд.Z *)
      MD893 AT %MD893 : UDINT := 16#00000000;  (* CDN[78].Tmax.(Ti |XYZ[0]): Темп. |Коорд.X *)
      MD894 AT %MD894 : UDINT := 16#00000000;  (* CDN[78].Tmax.(XYZ[1]|XYZ[2]): Коорд.Y|Коорд.Z *)
      MD895 AT %MD895 : UDINT := 16#00000000;  (* CDN[79].(ID|Tmid): Идент.|Tсред. *)
      MD896 AT %MD896 : UDINT := 16#00000000;  (* CDN[79].Tmin.(Ti |XYZ[0]): Темп. |Коорд.X *)
      MD897 AT %MD897 : UDINT := 16#00000000;  (* CDN[79].Tmin.(XYZ[1]|XYZ[2]): Коорд.Y|Коорд.Z *)
      MD898 AT %MD898 : UDINT := 16#00000000;  (* CDN[79].Tmax.(Ti |XYZ[0]): Темп. |Коорд.X *)
      MD899 AT %MD899 : UDINT := 16#00000000;  (* CDN[79].Tmax.(XYZ[1]|XYZ[2]): Коорд.Y|Коорд.Z *)
      MD900 AT %MD900 : UDINT := 16#00000000;  (* CDN[80].(ID|Tmid): Идент.|Tсред. *)
      MD901 AT %MD901 : UDINT := 16#00000000;  (* CDN[80].Tmin.(Ti |XYZ[0]): Темп. |Коорд.X *)
      MD902 AT %MD902 : UDINT := 16#00000000;  (* CDN[80].Tmin.(XYZ[1]|XYZ[2]): Коорд.Y|Коорд.Z *)
      MD903 AT %MD903 : UDINT := 16#00000000;  (* CDN[80].Tmax.(Ti |XYZ[0]): Темп. |Коорд.X *)
      MD904 AT %MD904 : UDINT := 16#00000000;  (* CDN[80].Tmax.(XYZ[1]|XYZ[2]): Коорд.Y|Коорд.Z *)
      MD905 AT %MD905 : UDINT := 16#00000000;  (* CDN[81].(ID|Tmid): Идент.|Tсред. *)
      MD906 AT %MD906 : UDINT := 16#00000000;  (* CDN[81].Tmin.(Ti |XYZ[0]): Темп. |Коорд.X *)
      MD907 AT %MD907 : UDINT := 16#00000000;  (* CDN[81].Tmin.(XYZ[1]|XYZ[2]): Коорд.Y|Коорд.Z *)
      MD908 AT %MD908 : UDINT := 16#00000000;  (* CDN[81].Tmax.(Ti |XYZ[0]): Темп. |Коорд.X *)
      MD909 AT %MD909 : UDINT := 16#00000000;  (* CDN[81].Tmax.(XYZ[1]|XYZ[2]): Коорд.Y|Коорд.Z *)
      MD910 AT %MD910 : UDINT := 16#00000000;  (* CDN[82].(ID|Tmid): Идент.|Tсред. *)
      MD911 AT %MD911 : UDINT := 16#00000000;  (* CDN[82].Tmin.(Ti |XYZ[0]): Темп. |Коорд.X *)
      MD912 AT %MD912 : UDINT := 16#00000000;  (* CDN[82].Tmin.(XYZ[1]|XYZ[2]): Коорд.Y|Коорд.Z *)
      MD913 AT %MD913 : UDINT := 16#00000000;  (* CDN[82].Tmax.(Ti |XYZ[0]): Темп. |Коорд.X *)
      MD914 AT %MD914 : UDINT := 16#00000000;  (* CDN[82].Tmax.(XYZ[1]|XYZ[2]): Коорд.Y|Коорд.Z *)
      MD915 AT %MD915 : UDINT := 16#00000000;  (* CDN[83].(ID|Tmid): Идент.|Tсред. *)
      MD916 AT %MD916 : UDINT := 16#00000000;  (* CDN[83].Tmin.(Ti |XYZ[0]): Темп. |Коорд.X *)
      MD917 AT %MD917 : UDINT := 16#00000000;  (* CDN[83].Tmin.(XYZ[1]|XYZ[2]): Коорд.Y|Коорд.Z *)
      MD918 AT %MD918 : UDINT := 16#00000000;  (* CDN[83].Tmax.(Ti |XYZ[0]): Темп. |Коорд.X *)
      MD919 AT %MD919 : UDINT := 16#00000000;  (* CDN[83].Tmax.(XYZ[1]|XYZ[2]): Коорд.Y|Коорд.Z *)
      MD920 AT %MD920 : UDINT := 16#00000000;  (* CDN[84].(ID|Tmid): Идент.|Tсред. *)
      MD921 AT %MD921 : UDINT := 16#00000000;  (* CDN[84].Tmin.(Ti |XYZ[0]): Темп. |Коорд.X *)
      MD922 AT %MD922 : UDINT := 16#00000000;  (* CDN[84].Tmin.(XYZ[1]|XYZ[2]): Коорд.Y|Коорд.Z *)
      MD923 AT %MD923 : UDINT := 16#00000000;  (* CDN[84].Tmax.(Ti |XYZ[0]): Темп. |Коорд.X *)
      MD924 AT %MD924 : UDINT := 16#00000000;  (* CDN[84].Tmax.(XYZ[1]|XYZ[2]): Коорд.Y|Коорд.Z *)
      MD925 AT %MD925 : UDINT := 16#00000000;  (* CDN[85].(ID|Tmid): Идент.|Tсред. *)
      MD926 AT %MD926 : UDINT := 16#00000000;  (* CDN[85].Tmin.(Ti |XYZ[0]): Темп. |Коорд.X *)
      MD927 AT %MD927 : UDINT := 16#00000000;  (* CDN[85].Tmin.(XYZ[1]|XYZ[2]): Коорд.Y|Коорд.Z *)
      MD928 AT %MD928 : UDINT := 16#00000000;  (* CDN[85].Tmax.(Ti |XYZ[0]): Темп. |Коорд.X *)
      MD929 AT %MD929 : UDINT := 16#00000000;  (* CDN[85].Tmax.(XYZ[1]|XYZ[2]): Коорд.Y|Коорд.Z *)
      MD930 AT %MD930 : UDINT := 16#00000000;  (* CDN[86].(ID|Tmid): Идент.|Tсред. *)
      MD931 AT %MD931 : UDINT := 16#00000000;  (* CDN[86].Tmin.(Ti |XYZ[0]): Темп. |Коорд.X *)
      MD932 AT %MD932 : UDINT := 16#00000000;  (* CDN[86].Tmin.(XYZ[1]|XYZ[2]): Коорд.Y|Коорд.Z *)
      MD933 AT %MD933 : UDINT := 16#00000000;  (* CDN[86].Tmax.(Ti |XYZ[0]): Темп. |Коорд.X *)
      MD934 AT %MD934 : UDINT := 16#00000000;  (* CDN[86].Tmax.(XYZ[1]|XYZ[2]): Коорд.Y|Коорд.Z *)
      MD935 AT %MD935 : UDINT := 16#00000000;  (* CDN[87].(ID|Tmid): Идент.|Tсред. *)
      MD936 AT %MD936 : UDINT := 16#00000000;  (* CDN[87].Tmin.(Ti |XYZ[0]): Темп. |Коорд.X *)
      MD937 AT %MD937 : UDINT := 16#00000000;  (* CDN[87].Tmin.(XYZ[1]|XYZ[2]): Коорд.Y|Коорд.Z *)
      MD938 AT %MD938 : UDINT := 16#00000000;  (* CDN[87].Tmax.(Ti |XYZ[0]): Темп. |Коорд.X *)
      MD939 AT %MD939 : UDINT := 16#00000000;  (* CDN[87].Tmax.(XYZ[1]|XYZ[2]): Коорд.Y|Коорд.Z *)
      MD940 AT %MD940 : UDINT := 16#00000000;  (* CDN[88].(ID|Tmid): Идент.|Tсред. *)
      MD941 AT %MD941 : UDINT := 16#00000000;  (* CDN[88].Tmin.(Ti |XYZ[0]): Темп. |Коорд.X *)
      MD942 AT %MD942 : UDINT := 16#00000000;  (* CDN[88].Tmin.(XYZ[1]|XYZ[2]): Коорд.Y|Коорд.Z *)
      MD943 AT %MD943 : UDINT := 16#00000000;  (* CDN[88].Tmax.(Ti |XYZ[0]): Темп. |Коорд.X *)
      MD944 AT %MD944 : UDINT := 16#00000000;  (* CDN[88].Tmax.(XYZ[1]|XYZ[2]): Коорд.Y|Коорд.Z *)
      MD945 AT %MD945 : UDINT := 16#00000000;  (* CDN[89].(ID|Tmid): Идент.|Tсред. *)
      MD946 AT %MD946 : UDINT := 16#00000000;  (* CDN[89].Tmin.(Ti |XYZ[0]): Темп. |Коорд.X *)
      MD947 AT %MD947 : UDINT := 16#00000000;  (* CDN[89].Tmin.(XYZ[1]|XYZ[2]): Коорд.Y|Коорд.Z *)
      MD948 AT %MD948 : UDINT := 16#00000000;  (* CDN[89].Tmax.(Ti |XYZ[0]): Темп. |Коорд.X *)
      MD949 AT %MD949 : UDINT := 16#00000000;  (* CDN[89].Tmax.(XYZ[1]|XYZ[2]): Коорд.Y|Коорд.Z *)
      MD950 AT %MD950 : UDINT := 16#00000000;  (* CDN[90].(ID|Tmid): Идент.|Tсред. *)
      MD951 AT %MD951 : UDINT := 16#00000000;  (* CDN[90].Tmin.(Ti |XYZ[0]): Темп. |Коорд.X *)
      MD952 AT %MD952 : UDINT := 16#00000000;  (* CDN[90].Tmin.(XYZ[1]|XYZ[2]): Коорд.Y|Коорд.Z *)
      MD953 AT %MD953 : UDINT := 16#00000000;  (* CDN[90].Tmax.(Ti |XYZ[0]): Темп. |Коорд.X *)
      MD954 AT %MD954 : UDINT := 16#00000000;  (* CDN[90].Tmax.(XYZ[1]|XYZ[2]): Коорд.Y|Коорд.Z *)
      MD955 AT %MD955 : UDINT := 16#00000000;  (* CDN[91].(ID|Tmid): Идент.|Tсред. *)
      MD956 AT %MD956 : UDINT := 16#00000000;  (* CDN[91].Tmin.(Ti |XYZ[0]): Темп. |Коорд.X *)
      MD957 AT %MD957 : UDINT := 16#00000000;  (* CDN[91].Tmin.(XYZ[1]|XYZ[2]): Коорд.Y|Коорд.Z *)
      MD958 AT %MD958 : UDINT := 16#00000000;  (* CDN[91].Tmax.(Ti |XYZ[0]): Темп. |Коорд.X *)
      MD959 AT %MD959 : UDINT := 16#00000000;  (* CDN[91].Tmax.(XYZ[1]|XYZ[2]): Коорд.Y|Коорд.Z *)
      MD960 AT %MD960 : UDINT := 16#00000000;  (* CDN[92].(ID|Tmid): Идент.|Tсред. *)
      MD961 AT %MD961 : UDINT := 16#00000000;  (* CDN[92].Tmin.(Ti |XYZ[0]): Темп. |Коорд.X *)
      MD962 AT %MD962 : UDINT := 16#00000000;  (* CDN[92].Tmin.(XYZ[1]|XYZ[2]): Коорд.Y|Коорд.Z *)
      MD963 AT %MD963 : UDINT := 16#00000000;  (* CDN[92].Tmax.(Ti |XYZ[0]): Темп. |Коорд.X *)
      MD964 AT %MD964 : UDINT := 16#00000000;  (* CDN[92].Tmax.(XYZ[1]|XYZ[2]): Коорд.Y|Коорд.Z *)
      MD965 AT %MD965 : UDINT := 16#00000000;  (* CDN[93].(ID|Tmid): Идент.|Tсред. *)
      MD966 AT %MD966 : UDINT := 16#00000000;  (* CDN[93].Tmin.(Ti |XYZ[0]): Темп. |Коорд.X *)
      MD967 AT %MD967 : UDINT := 16#00000000;  (* CDN[93].Tmin.(XYZ[1]|XYZ[2]): Коорд.Y|Коорд.Z *)
      MD968 AT %MD968 : UDINT := 16#00000000;  (* CDN[93].Tmax.(Ti |XYZ[0]): Темп. |Коорд.X *)
      MD969 AT %MD969 : UDINT := 16#00000000;  (* CDN[93].Tmax.(XYZ[1]|XYZ[2]): Коорд.Y|Коорд.Z *)
      MD970 AT %MD970 : UDINT := 16#00000000;  (* CDN[94].(ID|Tmid): Идент.|Tсред. *)
      MD971 AT %MD971 : UDINT := 16#00000000;  (* CDN[94].Tmin.(Ti |XYZ[0]): Темп. |Коорд.X *)
      MD972 AT %MD972 : UDINT := 16#00000000;  (* CDN[94].Tmin.(XYZ[1]|XYZ[2]): Коорд.Y|Коорд.Z *)
      MD973 AT %MD973 : UDINT := 16#00000000;  (* CDN[94].Tmax.(Ti |XYZ[0]): Темп. |Коорд.X *)
      MD974 AT %MD974 : UDINT := 16#00000000;  (* CDN[94].Tmax.(XYZ[1]|XYZ[2]): Коорд.Y|Коорд.Z *)
      MD975 AT %MD975 : UDINT := 16#00000000;  (* CDN[95].(ID|Tmid): Идент.|Tсред. *)
      MD976 AT %MD976 : UDINT := 16#00000000;  (* CDN[95].Tmin.(Ti |XYZ[0]): Темп. |Коорд.X *)
      MD977 AT %MD977 : UDINT := 16#00000000;  (* CDN[95].Tmin.(XYZ[1]|XYZ[2]): Коорд.Y|Коорд.Z *)
      MD978 AT %MD978 : UDINT := 16#00000000;  (* CDN[95].Tmax.(Ti |XYZ[0]): Темп. |Коорд.X *)
      MD979 AT %MD979 : UDINT := 16#00000000;  (* CDN[95].Tmax.(XYZ[1]|XYZ[2]): Коорд.Y|Коорд.Z *)
      MD980 AT %MD980 : UDINT := 16#00000000;  (* CDN[96].(ID|Tmid): Идент.|Tсред. *)
      MD981 AT %MD981 : UDINT := 16#00000000;  (* CDN[96].Tmin.(Ti |XYZ[0]): Темп. |Коорд.X *)
      MD982 AT %MD982 : UDINT := 16#00000000;  (* CDN[96].Tmin.(XYZ[1]|XYZ[2]): Коорд.Y|Коорд.Z *)
      MD983 AT %MD983 : UDINT := 16#00000000;  (* CDN[96].Tmax.(Ti |XYZ[0]): Темп. |Коорд.X *)
      MD984 AT %MD984 : UDINT := 16#00000000;  (* CDN[96].Tmax.(XYZ[1]|XYZ[2]): Коорд.Y|Коорд.Z *)
      MD985 AT %MD985 : UDINT := 16#00000000;  (* CDN[97].(ID|Tmid): Идент.|Tсред. *)
      MD986 AT %MD986 : UDINT := 16#00000000;  (* CDN[97].Tmin.(Ti |XYZ[0]): Темп. |Коорд.X *)
      MD987 AT %MD987 : UDINT := 16#00000000;  (* CDN[97].Tmin.(XYZ[1]|XYZ[2]): Коорд.Y|Коорд.Z *)
      MD988 AT %MD988 : UDINT := 16#00000000;  (* CDN[97].Tmax.(Ti |XYZ[0]): Темп. |Коорд.X *)
      MD989 AT %MD989 : UDINT := 16#00000000;  (* CDN[97].Tmax.(XYZ[1]|XYZ[2]): Коорд.Y|Коорд.Z *)
      MD990 AT %MD990 : UDINT := 16#00000000;  (* CDN[98].(ID|Tmid): Идент.|Tсред. *)
      MD991 AT %MD991 : UDINT := 16#00000000;  (* CDN[98].Tmin.(Ti |XYZ[0]): Темп. |Коорд.X *)
      MD992 AT %MD992 : UDINT := 16#00000000;  (* CDN[98].Tmin.(XYZ[1]|XYZ[2]): Коорд.Y|Коорд.Z *)
      MD993 AT %MD993 : UDINT := 16#00000000;  (* CDN[98].Tmax.(Ti |XYZ[0]): Темп. |Коорд.X *)
      MD994 AT %MD994 : UDINT := 16#00000000;  (* CDN[98].Tmax.(XYZ[1]|XYZ[2]): Коорд.Y|Коорд.Z *)
      MD995 AT %MD995 : UDINT := 16#00000000;  (* CDN[99].(ID|Tmid): Идент.|Tсред. *)
      MD996 AT %MD996 : UDINT := 16#00000000;  (* CDN[99].Tmin.(Ti |XYZ[0]): Темп. |Коорд.X *)
      MD997 AT %MD997 : UDINT := 16#00000000;  (* CDN[99].Tmin.(XYZ[1]|XYZ[2]): Коорд.Y|Коорд.Z *)
      MD998 AT %MD998 : UDINT := 16#00000000;  (* CDN[99].Tmax.(Ti |XYZ[0]): Темп. |Коорд.X *)
      MD999 AT %MD999 : UDINT := 16#00000000;  (* CDN[99].Tmax.(XYZ[1]|XYZ[2]): Коорд.Y|Коорд.Z *)
      MD1000 AT %MD1000 : UDINT := 16#00000000;  (* Резерв 0 *)
      MD1001 AT %MD1001 : UDINT := 16#00000000;  (* Резерв 1 *)
      MD1002 AT %MD1002 : UDINT := 16#00000000;  (* Резерв 2 *)
      MD1003 AT %MD1003 : UDINT := 16#00000000;  (* Резерв 3 *)
      MD1004 AT %MD1004 : UDINT := 16#00000000;  (* Резерв 4 *)
      MD1005 AT %MD1005 : UDINT := 16#00000000;  (* Резерв 5 *)
      MD1006 AT %MD1006 : UDINT := 16#00000000;  (* Резерв 6 *)
      MD1007 AT %MD1007 : UDINT := 16#00000000;  (* Резерв 7 *)
      MD1008 AT %MD1008 : UDINT := 16#00000000;  (* Резерв 8 *)
      MD1009 AT %MD1009 : UDINT := 16#00000000;  (* Резерв 9 *)
      MD1010 AT %MD1010 : UDINT := 16#00000000;  (* Резерв 10 *)
      MD1011 AT %MD1011 : UDINT := 16#00000000;  (* Резерв 11 *)
      MD1012 AT %MD1012 : UDINT := 16#00000000;  (* Резерв 12 *)
      MD1013 AT %MD1013 : UDINT := 16#00000000;  (* Резерв 13 *)
      MD1014 AT %MD1014 : UDINT := 16#00000000;  (* Резерв 14 *)
      MD1015 AT %MD1015 : UDINT := 16#00000000;  (* Резерв 15 *)
      MD1016 AT %MD1016 : UDINT := 16#00000000;  (* Резерв 16 *)
      MD1017 AT %MD1017 : UDINT := 16#00000000;  (* Резерв 17 *)
      MD1018 AT %MD1018 : UDINT := 16#00000000;  (* Резерв 18 *)
      MD1019 AT %MD1019 : UDINT := 16#00000000;  (* Резерв 19 *)
      MD1020 AT %MD1020 : UDINT := 16#00000000;  (* Резерв 20 *)
      MD1021 AT %MD1021 : UDINT := 16#00000000;  (* Резерв 21 *)
      MD1022 AT %MD1022 : UDINT := 16#00000000;  (* Резерв 22 *)
      MD1023 AT %MD1023 : UDINT := 16#00000000;  (* Резерв 23 *)
    END_VAR
    VAR_GLOBAL
      ML0 AT %ML0 : ULINT := 16#0123456789ABCDEF;  (* T3D[0]|T3D[1]|T3D[2]|T3D[3] *)
      ML1 AT %ML1 : ULINT := 16#0123456789ABCDEF;  (* T3D[4]|T3D[5]|T3D[6]|T3D[7] *)
      ML2 AT %ML2 : ULINT := 16#0123456789ABCDEF;  (* T3D[8]|T3D[9]|T3D[10]|T3D[11] *)
      ML3 AT %ML3 : ULINT := 16#0123456789ABCDEF;  (* T3D[12]|T3D[13]|T3D[14]|T3D[15] *)
      ML4 AT %ML4 : ULINT := 16#0123456789ABCDEF;  (* T3D[16]|T3D[17]|T3D[18]|T3D[19] *)
      ML5 AT %ML5 : ULINT := 16#0123456789ABCDEF;  (* T3D[20]|T3D[21]|T3D[22]|T3D[23] *)
      ML6 AT %ML6 : ULINT := 16#0123456789ABCDEF;  (* T3D[24]|T3D[25]|T3D[26]|T3D[27] *)
      ML7 AT %ML7 : ULINT := 16#0123456789ABCDEF;  (* T3D[28]|T3D[29]|T3D[30]|T3D[31] *)
      ML8 AT %ML8 : ULINT := 16#0123456789ABCDEF;  (* T3D[32]|T3D[33]|T3D[34]|T3D[35] *)
      ML9 AT %ML9 : ULINT := 16#0123456789ABCDEF;  (* T3D[36]|T3D[37]|T3D[38]|T3D[39] *)
      ML10 AT %ML10 : ULINT := 16#0123456789ABCDEF;  (* T3D[40]|T3D[41]|T3D[42]|T3D[43] *)
      ML11 AT %ML11 : ULINT := 16#0123456789ABCDEF;  (* T3D[44]|T3D[45]|T3D[46]|T3D[47] *)
      ML12 AT %ML12 : ULINT := 16#0123456789ABCDEF;  (* T3D[48]|T3D[49]|T3D[50]|T3D[51] *)
      ML13 AT %ML13 : ULINT := 16#0123456789ABCDEF;  (* T3D[52]|T3D[53]|T3D[54]|T3D[55] *)
      ML14 AT %ML14 : ULINT := 16#0123456789ABCDEF;  (* T3D[56]|T3D[57]|T3D[58]|T3D[59] *)
      ML15 AT %ML15 : ULINT := 16#0123456789ABCDEF;  (* T3D[60]|T3D[61]|T3D[62]|T3D[63] *)
      ML16 AT %ML16 : ULINT := 16#0123456789ABCDEF;  (* T3D[64]|T3D[65]|T3D[66]|T3D[67] *)
      ML17 AT %ML17 : ULINT := 16#0123456789ABCDEF;  (* T3D[68]|T3D[69]|T3D[70]|T3D[71] *)
      ML18 AT %ML18 : ULINT := 16#0123456789ABCDEF;  (* T3D[72]|T3D[73]|T3D[74]|T3D[75] *)
      ML19 AT %ML19 : ULINT := 16#0123456789ABCDEF;  (* T3D[76]|T3D[77]|T3D[78]|T3D[79] *)
      ML20 AT %ML20 : ULINT := 16#0123456789ABCDEF;  (* T3D[80]|T3D[81]|T3D[82]|T3D[83] *)
      ML21 AT %ML21 : ULINT := 16#0123456789ABCDEF;  (* T3D[84]|T3D[85]|T3D[86]|T3D[87] *)
      ML22 AT %ML22 : ULINT := 16#0123456789ABCDEF;  (* T3D[88]|T3D[89]|T3D[90]|T3D[91] *)
      ML23 AT %ML23 : ULINT := 16#0123456789ABCDEF;  (* T3D[92]|T3D[93]|T3D[94]|T3D[95] *)
      ML24 AT %ML24 : ULINT := 16#0123456789ABCDEF;  (* T3D[96]|T3D[97]|T3D[98]|T3D[99] *)
      ML25 AT %ML25 : ULINT := 16#0123456789ABCDEF;  (* T3D[100]|T3D[101]|T3D[102]|T3D[103] *)
      ML26 AT %ML26 : ULINT := 16#0123456789ABCDEF;  (* T3D[104]|T3D[105]|T3D[106]|T3D[107] *)
      ML27 AT %ML27 : ULINT := 16#0123456789ABCDEF;  (* T3D[108]|T3D[109]|T3D[110]|T3D[111] *)
      ML28 AT %ML28 : ULINT := 16#0123456789ABCDEF;  (* T3D[112]|T3D[113]|T3D[114]|T3D[115] *)
      ML29 AT %ML29 : ULINT := 16#0123456789ABCDEF;  (* T3D[116]|T3D[117]|T3D[118]|T3D[119] *)
      ML30 AT %ML30 : ULINT := 16#0123456789ABCDEF;  (* T3D[120]|T3D[121]|T3D[122]|T3D[123] *)
      ML31 AT %ML31 : ULINT := 16#0123456789ABCDEF;  (* T3D[124]|T3D[125]|T3D[126]|T3D[127] *)
      ML32 AT %ML32 : ULINT := 16#0123456789ABCDEF;  (* T3D[128]|T3D[129]|T3D[130]|T3D[131] *)
      ML33 AT %ML33 : ULINT := 16#0123456789ABCDEF;  (* T3D[132]|T3D[133]|T3D[134]|T3D[135] *)
      ML34 AT %ML34 : ULINT := 16#0123456789ABCDEF;  (* T3D[136]|T3D[137]|T3D[138]|T3D[139] *)
      ML35 AT %ML35 : ULINT := 16#0123456789ABCDEF;  (* T3D[140]|T3D[141]|T3D[142]|T3D[143] *)
      ML36 AT %ML36 : ULINT := 16#0123456789ABCDEF;  (* T3D[144]|T3D[145]|T3D[146]|T3D[147] *)
      ML37 AT %ML37 : ULINT := 16#0123456789ABCDEF;  (* T3D[148]|T3D[149]|T3D[150]|T3D[151] *)
      ML38 AT %ML38 : ULINT := 16#0123456789ABCDEF;  (* T3D[152]|T3D[153]|T3D[154]|T3D[155] *)
      ML39 AT %ML39 : ULINT := 16#0123456789ABCDEF;  (* T3D[156]|T3D[157]|T3D[158]|T3D[159] *)
      ML40 AT %ML40 : ULINT := 16#0123456789ABCDEF;  (* T3D[160]|T3D[161]|T3D[162]|T3D[163] *)
      ML41 AT %ML41 : ULINT := 16#0123456789ABCDEF;  (* T3D[164]|T3D[165]|T3D[166]|T3D[167] *)
      ML42 AT %ML42 : ULINT := 16#0123456789ABCDEF;  (* T3D[168]|T3D[169]|T3D[170]|T3D[171] *)
      ML43 AT %ML43 : ULINT := 16#0123456789ABCDEF;  (* T3D[172]|T3D[173]|T3D[174]|T3D[175] *)
      ML44 AT %ML44 : ULINT := 16#0123456789ABCDEF;  (* T3D[176]|T3D[177]|T3D[178]|T3D[179] *)
      ML45 AT %ML45 : ULINT := 16#0123456789ABCDEF;  (* T3D[180]|T3D[181]|T3D[182]|T3D[183] *)
      ML46 AT %ML46 : ULINT := 16#0123456789ABCDEF;  (* T3D[184]|T3D[185]|T3D[186]|T3D[187] *)
      ML47 AT %ML47 : ULINT := 16#0123456789ABCDEF;  (* T3D[188]|T3D[189]|T3D[190]|T3D[191] *)
      ML48 AT %ML48 : ULINT := 16#0123456789ABCDEF;  (* T3D[192]|T3D[193]|T3D[194]|T3D[195] *)
      ML49 AT %ML49 : ULINT := 16#0123456789ABCDEF;  (* T3D[196]|T3D[197]|T3D[198]|T3D[199] *)
      ML50 AT %ML50 : ULINT := 16#0123456789ABCDEF;  (* T3D[200]|T3D[201]|T3D[202]|T3D[203] *)
      ML51 AT %ML51 : ULINT := 16#0123456789ABCDEF;  (* T3D[204]|T3D[205]|T3D[206]|T3D[207] *)
      ML52 AT %ML52 : ULINT := 16#0123456789ABCDEF;  (* T3D[208]|T3D[209]|T3D[210]|T3D[211] *)
      ML53 AT %ML53 : ULINT := 16#0123456789ABCDEF;  (* T3D[212]|T3D[213]|T3D[214]|T3D[215] *)
      ML54 AT %ML54 : ULINT := 16#0123456789ABCDEF;  (* T3D[216]|T3D[217]|T3D[218]|T3D[219] *)
      ML55 AT %ML55 : ULINT := 16#0123456789ABCDEF;  (* T3D[220]|T3D[221]|T3D[222]|T3D[223] *)
      ML56 AT %ML56 : ULINT := 16#0123456789ABCDEF;  (* T3D[224]|T3D[225]|T3D[226]|T3D[227] *)
      ML57 AT %ML57 : ULINT := 16#0123456789ABCDEF;  (* T3D[228]|T3D[229]|T3D[230]|T3D[231] *)
      ML58 AT %ML58 : ULINT := 16#0123456789ABCDEF;  (* T3D[232]|T3D[233]|T3D[234]|T3D[235] *)
      ML59 AT %ML59 : ULINT := 16#0123456789ABCDEF;  (* T3D[236]|T3D[237]|T3D[238]|T3D[239] *)
      ML60 AT %ML60 : ULINT := 16#0123456789ABCDEF;  (* T3D[240]|T3D[241]|T3D[242]|T3D[243] *)
      ML61 AT %ML61 : ULINT := 16#0123456789ABCDEF;  (* T3D[244]|T3D[245]|T3D[246]|T3D[247] *)
      ML62 AT %ML62 : ULINT := 16#0123456789ABCDEF;  (* T3D[248]|T3D[249]|T3D[250]|T3D[251] *)
      ML63 AT %ML63 : ULINT := 16#0123456789ABCDEF;  (* T3D[252]|T3D[253]|T3D[254]|T3D[255] *)
      ML64 AT %ML64 : ULINT := 16#0123456789ABCDEF;  (* T3D[256]|T3D[257]|T3D[258]|T3D[259] *)
      ML65 AT %ML65 : ULINT := 16#0123456789ABCDEF;  (* T3D[260]|T3D[261]|T3D[262]|T3D[263] *)
      ML66 AT %ML66 : ULINT := 16#0123456789ABCDEF;  (* T3D[264]|T3D[265]|T3D[266]|T3D[267] *)
      ML67 AT %ML67 : ULINT := 16#0123456789ABCDEF;  (* T3D[268]|T3D[269]|T3D[270]|T3D[271] *)
      ML68 AT %ML68 : ULINT := 16#0123456789ABCDEF;  (* T3D[272]|T3D[273]|T3D[274]|T3D[275] *)
      ML69 AT %ML69 : ULINT := 16#0123456789ABCDEF;  (* T3D[276]|T3D[277]|T3D[278]|T3D[279] *)
      ML70 AT %ML70 : ULINT := 16#0123456789ABCDEF;  (* T3D[280]|T3D[281]|T3D[282]|T3D[283] *)
      ML71 AT %ML71 : ULINT := 16#0123456789ABCDEF;  (* T3D[284]|T3D[285]|T3D[286]|T3D[287] *)
      ML72 AT %ML72 : ULINT := 16#0123456789ABCDEF;  (* T3D[288]|T3D[289]|T3D[290]|T3D[291] *)
      ML73 AT %ML73 : ULINT := 16#0123456789ABCDEF;  (* T3D[292]|T3D[293]|T3D[294]|T3D[295] *)
      ML74 AT %ML74 : ULINT := 16#0123456789ABCDEF;  (* T3D[296]|T3D[297]|T3D[298]|T3D[299] *)
      ML75 AT %ML75 : ULINT := 16#0123456789ABCDEF;  (* T3D[300]|T3D[301]|T3D[302]|T3D[303] *)
      ML76 AT %ML76 : ULINT := 16#0123456789ABCDEF;  (* T3D[304]|T3D[305]|T3D[306]|T3D[307] *)
      ML77 AT %ML77 : ULINT := 16#0123456789ABCDEF;  (* T3D[308]|T3D[309]|T3D[310]|T3D[311] *)
      ML78 AT %ML78 : ULINT := 16#0123456789ABCDEF;  (* T3D[312]|T3D[313]|T3D[314]|T3D[315] *)
      ML79 AT %ML79 : ULINT := 16#0123456789ABCDEF;  (* T3D[316]|T3D[317]|T3D[318]|T3D[319] *)
      ML80 AT %ML80 : ULINT := 16#0123456789ABCDEF;  (* T3D[320]|T3D[321]|T3D[322]|T3D[323] *)
      ML81 AT %ML81 : ULINT := 16#0123456789ABCDEF;  (* T3D[324]|T3D[325]|T3D[326]|T3D[327] *)
      ML82 AT %ML82 : ULINT := 16#0123456789ABCDEF;  (* T3D[328]|T3D[329]|T3D[330]|T3D[331] *)
      ML83 AT %ML83 : ULINT := 16#0123456789ABCDEF;  (* T3D[332]|T3D[333]|T3D[334]|T3D[335] *)
      ML84 AT %ML84 : ULINT := 16#0123456789ABCDEF;  (* T3D[336]|T3D[337]|T3D[338]|T3D[339] *)
      ML85 AT %ML85 : ULINT := 16#0123456789ABCDEF;  (* T3D[340]|T3D[341]|T3D[342]|T3D[343] *)
      ML86 AT %ML86 : ULINT := 16#0123456789ABCDEF;  (* T3D[344]|T3D[345]|T3D[346]|T3D[347] *)
      ML87 AT %ML87 : ULINT := 16#0123456789ABCDEF;  (* T3D[348]|T3D[349]|T3D[350]|T3D[351] *)
      ML88 AT %ML88 : ULINT := 16#0123456789ABCDEF;  (* T3D[352]|T3D[353]|T3D[354]|T3D[355] *)
      ML89 AT %ML89 : ULINT := 16#0123456789ABCDEF;  (* T3D[356]|T3D[357]|T3D[358]|T3D[359] *)
      ML90 AT %ML90 : ULINT := 16#0123456789ABCDEF;  (* T3D[360]|T3D[361]|T3D[362]|T3D[363] *)
      ML91 AT %ML91 : ULINT := 16#0123456789ABCDEF;  (* T3D[364]|T3D[365]|T3D[366]|T3D[367] *)
      ML92 AT %ML92 : ULINT := 16#0123456789ABCDEF;  (* T3D[368]|T3D[369]|T3D[370]|T3D[371] *)
      ML93 AT %ML93 : ULINT := 16#0123456789ABCDEF;  (* T3D[372]|T3D[373]|T3D[374]|T3D[375] *)
      ML94 AT %ML94 : ULINT := 16#0123456789ABCDEF;  (* T3D[376]|T3D[377]|T3D[378]|T3D[379] *)
      ML95 AT %ML95 : ULINT := 16#0123456789ABCDEF;  (* T3D[380]|T3D[381]|T3D[382]|T3D[383] *)
      ML96 AT %ML96 : ULINT := 16#0123456789ABCDEF;  (* T3D[384]|T3D[385]|T3D[386]|T3D[387] *)
      ML97 AT %ML97 : ULINT := 16#0123456789ABCDEF;  (* T3D[388]|T3D[389]|T3D[390]|T3D[391] *)
      ML98 AT %ML98 : ULINT := 16#0123456789ABCDEF;  (* T3D[392]|T3D[393]|T3D[394]|T3D[395] *)
      ML99 AT %ML99 : ULINT := 16#0123456789ABCDEF;  (* T3D[396]|T3D[397]|T3D[398]|T3D[399] *)
      ML100 AT %ML100 : ULINT := 16#0123456789ABCDEF;  (* T3D[400]|T3D[401]|T3D[402]|T3D[403] *)
      ML101 AT %ML101 : ULINT := 16#0123456789ABCDEF;  (* T3D[404]|T3D[405]|T3D[406]|T3D[407] *)
      ML102 AT %ML102 : ULINT := 16#0123456789ABCDEF;  (* T3D[408]|T3D[409]|T3D[410]|T3D[411] *)
      ML103 AT %ML103 : ULINT := 16#0123456789ABCDEF;  (* T3D[412]|T3D[413]|T3D[414]|T3D[415] *)
      ML104 AT %ML104 : ULINT := 16#0123456789ABCDEF;  (* T3D[416]|T3D[417]|T3D[418]|T3D[419] *)
      ML105 AT %ML105 : ULINT := 16#0123456789ABCDEF;  (* T3D[420]|T3D[421]|T3D[422]|T3D[423] *)
      ML106 AT %ML106 : ULINT := 16#0123456789ABCDEF;  (* T3D[424]|T3D[425]|T3D[426]|T3D[427] *)
      ML107 AT %ML107 : ULINT := 16#0123456789ABCDEF;  (* T3D[428]|T3D[429]|T3D[430]|T3D[431] *)
      ML108 AT %ML108 : ULINT := 16#0123456789ABCDEF;  (* T3D[432]|T3D[433]|T3D[434]|T3D[435] *)
      ML109 AT %ML109 : ULINT := 16#0123456789ABCDEF;  (* T3D[436]|T3D[437]|T3D[438]|T3D[439] *)
      ML110 AT %ML110 : ULINT := 16#0123456789ABCDEF;  (* T3D[440]|T3D[441]|T3D[442]|T3D[443] *)
      ML111 AT %ML111 : ULINT := 16#0123456789ABCDEF;  (* T3D[444]|T3D[445]|T3D[446]|T3D[447] *)
      ML112 AT %ML112 : ULINT := 16#0123456789ABCDEF;  (* T3D[448]|T3D[449]|T3D[450]|T3D[451] *)
      ML113 AT %ML113 : ULINT := 16#0123456789ABCDEF;  (* T3D[452]|T3D[453]|T3D[454]|T3D[455] *)
      ML114 AT %ML114 : ULINT := 16#0123456789ABCDEF;  (* T3D[456]|T3D[457]|T3D[458]|T3D[459] *)
      ML115 AT %ML115 : ULINT := 16#0123456789ABCDEF;  (* T3D[460]|T3D[461]|T3D[462]|T3D[463] *)
      ML116 AT %ML116 : ULINT := 16#0123456789ABCDEF;  (* T3D[464]|T3D[465]|T3D[466]|T3D[467] *)
      ML117 AT %ML117 : ULINT := 16#0123456789ABCDEF;  (* T3D[468]|T3D[469]|T3D[470]|T3D[471] *)
      ML118 AT %ML118 : ULINT := 16#0123456789ABCDEF;  (* T3D[472]|T3D[473]|T3D[474]|T3D[475] *)
      ML119 AT %ML119 : ULINT := 16#0123456789ABCDEF;  (* T3D[476]|T3D[477]|T3D[478]|T3D[479] *)
      ML120 AT %ML120 : ULINT := 16#0123456789ABCDEF;  (* T3D[480]|T3D[481]|T3D[482]|T3D[483] *)
      ML121 AT %ML121 : ULINT := 16#0123456789ABCDEF;  (* T3D[484]|T3D[485]|T3D[486]|T3D[487] *)
      ML122 AT %ML122 : ULINT := 16#0123456789ABCDEF;  (* T3D[488]|T3D[489]|T3D[490]|T3D[491] *)
      ML123 AT %ML123 : ULINT := 16#0123456789ABCDEF;  (* T3D[492]|T3D[493]|T3D[494]|T3D[495] *)
      ML124 AT %ML124 : ULINT := 16#0123456789ABCDEF;  (* T3D[496]|T3D[497]|T3D[498]|T3D[499] *)
      ML125 AT %ML125 : ULINT := 16#0123456789ABCDEF;  (* T3D[500]|T3D[501]|T3D[502]|T3D[503] *)
      ML126 AT %ML126 : ULINT := 16#0123456789ABCDEF;  (* T3D[504]|T3D[505]|T3D[506]|T3D[507] *)
      ML127 AT %ML127 : ULINT := 16#0123456789ABCDEF;  (* T3D[508]|T3D[509]|T3D[510]|T3D[511] *)
      ML128 AT %ML128 : ULINT := 16#0123456789ABCDEF;  (* T3D[512]|T3D[513]|T3D[514]|T3D[515] *)
      ML129 AT %ML129 : ULINT := 16#0123456789ABCDEF;  (* T3D[516]|T3D[517]|T3D[518]|T3D[519] *)
      ML130 AT %ML130 : ULINT := 16#0123456789ABCDEF;  (* T3D[520]|T3D[521]|T3D[522]|T3D[523] *)
      ML131 AT %ML131 : ULINT := 16#0123456789ABCDEF;  (* T3D[524]|T3D[525]|T3D[526]|T3D[527] *)
      ML132 AT %ML132 : ULINT := 16#0123456789ABCDEF;  (* T3D[528]|T3D[529]|T3D[530]|T3D[531] *)
      ML133 AT %ML133 : ULINT := 16#0123456789ABCDEF;  (* T3D[532]|T3D[533]|T3D[534]|T3D[535] *)
      ML134 AT %ML134 : ULINT := 16#0123456789ABCDEF;  (* T3D[536]|T3D[537]|T3D[538]|T3D[539] *)
      ML135 AT %ML135 : ULINT := 16#0123456789ABCDEF;  (* T3D[540]|T3D[541]|T3D[542]|T3D[543] *)
      ML136 AT %ML136 : ULINT := 16#0123456789ABCDEF;  (* T3D[544]|T3D[545]|T3D[546]|T3D[547] *)
      ML137 AT %ML137 : ULINT := 16#0123456789ABCDEF;  (* T3D[548]|T3D[549]|T3D[550]|T3D[551] *)
      ML138 AT %ML138 : ULINT := 16#0123456789ABCDEF;  (* T3D[552]|T3D[553]|T3D[554]|T3D[555] *)
      ML139 AT %ML139 : ULINT := 16#0123456789ABCDEF;  (* T3D[556]|T3D[557]|T3D[558]|T3D[559] *)
      ML140 AT %ML140 : ULINT := 16#0123456789ABCDEF;  (* T3D[560]|T3D[561]|T3D[562]|T3D[563] *)
      ML141 AT %ML141 : ULINT := 16#0123456789ABCDEF;  (* T3D[564]|T3D[565]|T3D[566]|T3D[567] *)
      ML142 AT %ML142 : ULINT := 16#0123456789ABCDEF;  (* T3D[568]|T3D[569]|T3D[570]|T3D[571] *)
      ML143 AT %ML143 : ULINT := 16#0123456789ABCDEF;  (* T3D[572]|T3D[573]|T3D[574]|T3D[575] *)
      ML144 AT %ML144 : ULINT := 16#0123456789ABCDEF;  (* T3D[576]|T3D[577]|T3D[578]|T3D[579] *)
      ML145 AT %ML145 : ULINT := 16#0123456789ABCDEF;  (* T3D[580]|T3D[581]|T3D[582]|T3D[583] *)
      ML146 AT %ML146 : ULINT := 16#0123456789ABCDEF;  (* T3D[584]|T3D[585]|T3D[586]|T3D[587] *)
      ML147 AT %ML147 : ULINT := 16#0123456789ABCDEF;  (* T3D[588]|T3D[589]|T3D[590]|T3D[591] *)
      ML148 AT %ML148 : ULINT := 16#0123456789ABCDEF;  (* T3D[592]|T3D[593]|T3D[594]|T3D[595] *)
      ML149 AT %ML149 : ULINT := 16#0123456789ABCDEF;  (* T3D[596]|T3D[597]|T3D[598]|T3D[599] *)
      ML150 AT %ML150 : ULINT := 16#0123456789ABCDEF;  (* T3D[600]|T3D[601]|T3D[602]|T3D[603] *)
      ML151 AT %ML151 : ULINT := 16#0123456789ABCDEF;  (* T3D[604]|T3D[605]|T3D[606]|T3D[607] *)
      ML152 AT %ML152 : ULINT := 16#0123456789ABCDEF;  (* T3D[608]|T3D[609]|T3D[610]|T3D[611] *)
      ML153 AT %ML153 : ULINT := 16#0123456789ABCDEF;  (* T3D[612]|T3D[613]|T3D[614]|T3D[615] *)
      ML154 AT %ML154 : ULINT := 16#0123456789ABCDEF;  (* T3D[616]|T3D[617]|T3D[618]|T3D[619] *)
      ML155 AT %ML155 : ULINT := 16#0123456789ABCDEF;  (* T3D[620]|T3D[621]|T3D[622]|T3D[623] *)
      ML156 AT %ML156 : ULINT := 16#0123456789ABCDEF;  (* T3D[624]|T3D[625]|T3D[626]|T3D[627] *)
      ML157 AT %ML157 : ULINT := 16#0123456789ABCDEF;  (* T3D[628]|T3D[629]|T3D[630]|T3D[631] *)
      ML158 AT %ML158 : ULINT := 16#0123456789ABCDEF;  (* T3D[632]|T3D[633]|T3D[634]|T3D[635] *)
      ML159 AT %ML159 : ULINT := 16#0123456789ABCDEF;  (* T3D[636]|T3D[637]|T3D[638]|T3D[639] *)
      ML160 AT %ML160 : ULINT := 16#0123456789ABCDEF;  (* T3D[640]|T3D[641]|T3D[642]|T3D[643] *)
      ML161 AT %ML161 : ULINT := 16#0123456789ABCDEF;  (* T3D[644]|T3D[645]|T3D[646]|T3D[647] *)
      ML162 AT %ML162 : ULINT := 16#0123456789ABCDEF;  (* T3D[648]|T3D[649]|T3D[650]|T3D[651] *)
      ML163 AT %ML163 : ULINT := 16#0123456789ABCDEF;  (* T3D[652]|T3D[653]|T3D[654]|T3D[655] *)
      ML164 AT %ML164 : ULINT := 16#0123456789ABCDEF;  (* T3D[656]|T3D[657]|T3D[658]|T3D[659] *)
      ML165 AT %ML165 : ULINT := 16#0123456789ABCDEF;  (* T3D[660]|T3D[661]|T3D[662]|T3D[663] *)
      ML166 AT %ML166 : ULINT := 16#0123456789ABCDEF;  (* T3D[664]|T3D[665]|T3D[666]|T3D[667] *)
      ML167 AT %ML167 : ULINT := 16#0123456789ABCDEF;  (* T3D[668]|T3D[669]|T3D[670]|T3D[671] *)
      ML168 AT %ML168 : ULINT := 16#0123456789ABCDEF;  (* T3D[672]|T3D[673]|T3D[674]|T3D[675] *)
      ML169 AT %ML169 : ULINT := 16#0123456789ABCDEF;  (* T3D[676]|T3D[677]|T3D[678]|T3D[679] *)
      ML170 AT %ML170 : ULINT := 16#0123456789ABCDEF;  (* T3D[680]|T3D[681]|T3D[682]|T3D[683] *)
      ML171 AT %ML171 : ULINT := 16#0123456789ABCDEF;  (* T3D[684]|T3D[685]|T3D[686]|T3D[687] *)
      ML172 AT %ML172 : ULINT := 16#0123456789ABCDEF;  (* T3D[688]|T3D[689]|T3D[690]|T3D[691] *)
      ML173 AT %ML173 : ULINT := 16#0123456789ABCDEF;  (* T3D[692]|T3D[693]|T3D[694]|T3D[695] *)
      ML174 AT %ML174 : ULINT := 16#0123456789ABCDEF;  (* T3D[696]|T3D[697]|T3D[698]|T3D[699] *)
      ML175 AT %ML175 : ULINT := 16#0123456789ABCDEF;  (* T3D[700]|T3D[701]|T3D[702]|T3D[703] *)
      ML176 AT %ML176 : ULINT := 16#0123456789ABCDEF;  (* T3D[704]|T3D[705]|T3D[706]|T3D[707] *)
      ML177 AT %ML177 : ULINT := 16#0123456789ABCDEF;  (* T3D[708]|T3D[709]|T3D[710]|T3D[711] *)
      ML178 AT %ML178 : ULINT := 16#0123456789ABCDEF;  (* T3D[712]|T3D[713]|T3D[714]|T3D[715] *)
      ML179 AT %ML179 : ULINT := 16#0123456789ABCDEF;  (* T3D[716]|T3D[717]|T3D[718]|T3D[719] *)
      ML180 AT %ML180 : ULINT := 16#0123456789ABCDEF;  (* T3D[720]|T3D[721]|T3D[722]|T3D[723] *)
      ML181 AT %ML181 : ULINT := 16#0123456789ABCDEF;  (* T3D[724]|T3D[725]|T3D[726]|T3D[727] *)
      ML182 AT %ML182 : ULINT := 16#0123456789ABCDEF;  (* T3D[728]|T3D[729]|T3D[730]|T3D[731] *)
      ML183 AT %ML183 : ULINT := 16#0123456789ABCDEF;  (* T3D[732]|T3D[733]|T3D[734]|T3D[735] *)
      ML184 AT %ML184 : ULINT := 16#0123456789ABCDEF;  (* T3D[736]|T3D[737]|T3D[738]|T3D[739] *)
      ML185 AT %ML185 : ULINT := 16#0123456789ABCDEF;  (* T3D[740]|T3D[741]|T3D[742]|T3D[743] *)
      ML186 AT %ML186 : ULINT := 16#0123456789ABCDEF;  (* T3D[744]|T3D[745]|T3D[746]|T3D[747] *)
      ML187 AT %ML187 : ULINT := 16#0123456789ABCDEF;  (* T3D[748]|T3D[749]|T3D[750]|T3D[751] *)
      ML188 AT %ML188 : ULINT := 16#0123456789ABCDEF;  (* T3D[752]|T3D[753]|T3D[754]|T3D[755] *)
      ML189 AT %ML189 : ULINT := 16#0123456789ABCDEF;  (* T3D[756]|T3D[757]|T3D[758]|T3D[759] *)
      ML190 AT %ML190 : ULINT := 16#0123456789ABCDEF;  (* T3D[760]|T3D[761]|T3D[762]|T3D[763] *)
      ML191 AT %ML191 : ULINT := 16#0123456789ABCDEF;  (* T3D[764]|T3D[765]|T3D[766]|T3D[767] *)
      ML192 AT %ML192 : ULINT := 16#0123456789ABCDEF;  (* T3D[768]|T3D[769]|T3D[770]|T3D[771] *)
      ML193 AT %ML193 : ULINT := 16#0123456789ABCDEF;  (* T3D[772]|T3D[773]|T3D[774]|T3D[775] *)
      ML194 AT %ML194 : ULINT := 16#0123456789ABCDEF;  (* T3D[776]|T3D[777]|T3D[778]|T3D[779] *)
      ML195 AT %ML195 : ULINT := 16#0123456789ABCDEF;  (* T3D[780]|T3D[781]|T3D[782]|T3D[783] *)
      ML196 AT %ML196 : ULINT := 16#0123456789ABCDEF;  (* T3D[784]|T3D[785]|T3D[786]|T3D[787] *)
      ML197 AT %ML197 : ULINT := 16#0123456789ABCDEF;  (* T3D[788]|T3D[789]|T3D[790]|T3D[791] *)
      ML198 AT %ML198 : ULINT := 16#0123456789ABCDEF;  (* T3D[792]|T3D[793]|T3D[794]|T3D[795] *)
      ML199 AT %ML199 : ULINT := 16#0123456789ABCDEF;  (* T3D[796]|T3D[797]|T3D[798]|T3D[799] *)
      ML200 AT %ML200 : ULINT := 16#0123456789ABCDEF;  (* T3D[800]|T3D[801]|T3D[802]|T3D[803] *)
      ML201 AT %ML201 : ULINT := 16#0123456789ABCDEF;  (* T3D[804]|T3D[805]|T3D[806]|T3D[807] *)
      ML202 AT %ML202 : ULINT := 16#0123456789ABCDEF;  (* T3D[808]|T3D[809]|T3D[810]|T3D[811] *)
      ML203 AT %ML203 : ULINT := 16#0123456789ABCDEF;  (* T3D[812]|T3D[813]|T3D[814]|T3D[815] *)
      ML204 AT %ML204 : ULINT := 16#0123456789ABCDEF;  (* T3D[816]|T3D[817]|T3D[818]|T3D[819] *)
      ML205 AT %ML205 : ULINT := 16#0123456789ABCDEF;  (* T3D[820]|T3D[821]|T3D[822]|T3D[823] *)
      ML206 AT %ML206 : ULINT := 16#0123456789ABCDEF;  (* T3D[824]|T3D[825]|T3D[826]|T3D[827] *)
      ML207 AT %ML207 : ULINT := 16#0123456789ABCDEF;  (* T3D[828]|T3D[829]|T3D[830]|T3D[831] *)
      ML208 AT %ML208 : ULINT := 16#0123456789ABCDEF;  (* T3D[832]|T3D[833]|T3D[834]|T3D[835] *)
      ML209 AT %ML209 : ULINT := 16#0123456789ABCDEF;  (* T3D[836]|T3D[837]|T3D[838]|T3D[839] *)
      ML210 AT %ML210 : ULINT := 16#0123456789ABCDEF;  (* T3D[840]|T3D[841]|T3D[842]|T3D[843] *)
      ML211 AT %ML211 : ULINT := 16#0123456789ABCDEF;  (* T3D[844]|T3D[845]|T3D[846]|T3D[847] *)
      ML212 AT %ML212 : ULINT := 16#0123456789ABCDEF;  (* T3D[848]|T3D[849]|T3D[850]|T3D[851] *)
      ML213 AT %ML213 : ULINT := 16#0123456789ABCDEF;  (* T3D[852]|T3D[853]|T3D[854]|T3D[855] *)
      ML214 AT %ML214 : ULINT := 16#0123456789ABCDEF;  (* T3D[856]|T3D[857]|T3D[858]|T3D[859] *)
      ML215 AT %ML215 : ULINT := 16#0123456789ABCDEF;  (* T3D[860]|T3D[861]|T3D[862]|T3D[863] *)
      ML216 AT %ML216 : ULINT := 16#0123456789ABCDEF;  (* T3D[864]|T3D[865]|T3D[866]|T3D[867] *)
      ML217 AT %ML217 : ULINT := 16#0123456789ABCDEF;  (* T3D[868]|T3D[869]|T3D[870]|T3D[871] *)
      ML218 AT %ML218 : ULINT := 16#0123456789ABCDEF;  (* T3D[872]|T3D[873]|T3D[874]|T3D[875] *)
      ML219 AT %ML219 : ULINT := 16#0123456789ABCDEF;  (* T3D[876]|T3D[877]|T3D[878]|T3D[879] *)
      ML220 AT %ML220 : ULINT := 16#0123456789ABCDEF;  (* T3D[880]|T3D[881]|T3D[882]|T3D[883] *)
      ML221 AT %ML221 : ULINT := 16#0123456789ABCDEF;  (* T3D[884]|T3D[885]|T3D[886]|T3D[887] *)
      ML222 AT %ML222 : ULINT := 16#0123456789ABCDEF;  (* T3D[888]|T3D[889]|T3D[890]|T3D[891] *)
      ML223 AT %ML223 : ULINT := 16#0123456789ABCDEF;  (* T3D[892]|T3D[893]|T3D[894]|T3D[895] *)
      ML224 AT %ML224 : ULINT := 16#0123456789ABCDEF;  (* T3D[896]|T3D[897]|T3D[898]|T3D[899] *)
      ML225 AT %ML225 : ULINT := 16#0123456789ABCDEF;  (* T3D[900]|T3D[901]|T3D[902]|T3D[903] *)
      ML226 AT %ML226 : ULINT := 16#0123456789ABCDEF;  (* T3D[904]|T3D[905]|T3D[906]|T3D[907] *)
      ML227 AT %ML227 : ULINT := 16#0123456789ABCDEF;  (* T3D[908]|T3D[909]|T3D[910]|T3D[911] *)
      ML228 AT %ML228 : ULINT := 16#0123456789ABCDEF;  (* T3D[912]|T3D[913]|T3D[914]|T3D[915] *)
      ML229 AT %ML229 : ULINT := 16#0123456789ABCDEF;  (* T3D[916]|T3D[917]|T3D[918]|T3D[919] *)
      ML230 AT %ML230 : ULINT := 16#0123456789ABCDEF;  (* T3D[920]|T3D[921]|T3D[922]|T3D[923] *)
      ML231 AT %ML231 : ULINT := 16#0123456789ABCDEF;  (* T3D[924]|T3D[925]|T3D[926]|T3D[927] *)
      ML232 AT %ML232 : ULINT := 16#0123456789ABCDEF;  (* T3D[928]|T3D[929]|T3D[930]|T3D[931] *)
      ML233 AT %ML233 : ULINT := 16#0123456789ABCDEF;  (* T3D[932]|T3D[933]|T3D[934]|T3D[935] *)
      ML234 AT %ML234 : ULINT := 16#0123456789ABCDEF;  (* T3D[936]|T3D[937]|T3D[938]|T3D[939] *)
      ML235 AT %ML235 : ULINT := 16#0123456789ABCDEF;  (* T3D[940]|T3D[941]|T3D[942]|T3D[943] *)
      ML236 AT %ML236 : ULINT := 16#0123456789ABCDEF;  (* T3D[944]|T3D[945]|T3D[946]|T3D[947] *)
      ML237 AT %ML237 : ULINT := 16#0123456789ABCDEF;  (* T3D[948]|T3D[949]|T3D[950]|T3D[951] *)
      ML238 AT %ML238 : ULINT := 16#0123456789ABCDEF;  (* T3D[952]|T3D[953]|T3D[954]|T3D[955] *)
      ML239 AT %ML239 : ULINT := 16#0123456789ABCDEF;  (* T3D[956]|T3D[957]|T3D[958]|T3D[959] *)
      ML240 AT %ML240 : ULINT := 16#0123456789ABCDEF;  (* T3D[960]|T3D[961]|T3D[962]|T3D[963] *)
      ML241 AT %ML241 : ULINT := 16#0123456789ABCDEF;  (* T3D[964]|T3D[965]|T3D[966]|T3D[967] *)
      ML242 AT %ML242 : ULINT := 16#0123456789ABCDEF;  (* T3D[968]|T3D[969]|T3D[970]|T3D[971] *)
      ML243 AT %ML243 : ULINT := 16#0123456789ABCDEF;  (* T3D[972]|T3D[973]|T3D[974]|T3D[975] *)
      ML244 AT %ML244 : ULINT := 16#0123456789ABCDEF;  (* T3D[976]|T3D[977]|T3D[978]|T3D[979] *)
      ML245 AT %ML245 : ULINT := 16#0123456789ABCDEF;  (* T3D[980]|T3D[981]|T3D[982]|T3D[983] *)
      ML246 AT %ML246 : ULINT := 16#0123456789ABCDEF;  (* T3D[984]|T3D[985]|T3D[986]|T3D[987] *)
      ML247 AT %ML247 : ULINT := 16#0123456789ABCDEF;  (* T3D[988]|T3D[989]|T3D[990]|T3D[991] *)
      ML248 AT %ML248 : ULINT := 16#0123456789ABCDEF;  (* T3D[992]|T3D[993]|T3D[994]|T3D[995] *)
      ML249 AT %ML249 : ULINT := 16#0123456789ABCDEF;  (* T3D[996]|T3D[997]|T3D[998]|T3D[999] *)
      ML250 AT %ML250 : ULINT := 16#0123456789ABCDEF;  (* T3D[1000]|T3D[1001]|T3D[1002]|T3D[1003] *)
      ML251 AT %ML251 : ULINT := 16#0123456789ABCDEF;  (* T3D[1004]|T3D[1005]|T3D[1006]|T3D[1007] *)
      ML252 AT %ML252 : ULINT := 16#0123456789ABCDEF;  (* T3D[1008]|T3D[1009]|T3D[1010]|T3D[1011] *)
      ML253 AT %ML253 : ULINT := 16#0123456789ABCDEF;  (* T3D[1012]|T3D[1013]|T3D[1014]|T3D[1015] *)
      ML254 AT %ML254 : ULINT := 16#0123456789ABCDEF;  (* T3D[1016]|T3D[1017]|T3D[1018]|T3D[1019] *)
      ML255 AT %ML255 : ULINT := 16#0123456789ABCDEF;  (* T3D[1020]|T3D[1021]|T3D[1022]|T3D[1023] *)
      ML256 AT %ML256 : ULINT := 16#0123456789ABCDEF;  (* T3D[1024]|T3D[1025]|T3D[1026]|T3D[1027] *)
      ML257 AT %ML257 : ULINT := 16#0123456789ABCDEF;  (* T3D[1028]|T3D[1029]|T3D[1030]|T3D[1031] *)
      ML258 AT %ML258 : ULINT := 16#0123456789ABCDEF;  (* T3D[1032]|T3D[1033]|T3D[1034]|T3D[1035] *)
      ML259 AT %ML259 : ULINT := 16#0123456789ABCDEF;  (* T3D[1036]|T3D[1037]|T3D[1038]|T3D[1039] *)
      ML260 AT %ML260 : ULINT := 16#0123456789ABCDEF;  (* T3D[1040]|T3D[1041]|T3D[1042]|T3D[1043] *)
      ML261 AT %ML261 : ULINT := 16#0123456789ABCDEF;  (* T3D[1044]|T3D[1045]|T3D[1046]|T3D[1047] *)
      ML262 AT %ML262 : ULINT := 16#0123456789ABCDEF;  (* T3D[1048]|T3D[1049]|T3D[1050]|T3D[1051] *)
      ML263 AT %ML263 : ULINT := 16#0123456789ABCDEF;  (* T3D[1052]|T3D[1053]|T3D[1054]|T3D[1055] *)
      ML264 AT %ML264 : ULINT := 16#0123456789ABCDEF;  (* T3D[1056]|T3D[1057]|T3D[1058]|T3D[1059] *)
      ML265 AT %ML265 : ULINT := 16#0123456789ABCDEF;  (* T3D[1060]|T3D[1061]|T3D[1062]|T3D[1063] *)
      ML266 AT %ML266 : ULINT := 16#0123456789ABCDEF;  (* T3D[1064]|T3D[1065]|T3D[1066]|T3D[1067] *)
      ML267 AT %ML267 : ULINT := 16#0123456789ABCDEF;  (* T3D[1068]|T3D[1069]|T3D[1070]|T3D[1071] *)
      ML268 AT %ML268 : ULINT := 16#0123456789ABCDEF;  (* T3D[1072]|T3D[1073]|T3D[1074]|T3D[1075] *)
      ML269 AT %ML269 : ULINT := 16#0123456789ABCDEF;  (* T3D[1076]|T3D[1077]|T3D[1078]|T3D[1079] *)
      ML270 AT %ML270 : ULINT := 16#0123456789ABCDEF;  (* T3D[1080]|T3D[1081]|T3D[1082]|T3D[1083] *)
      ML271 AT %ML271 : ULINT := 16#0123456789ABCDEF;  (* T3D[1084]|T3D[1085]|T3D[1086]|T3D[1087] *)
      ML272 AT %ML272 : ULINT := 16#0123456789ABCDEF;  (* T3D[1088]|T3D[1089]|T3D[1090]|T3D[1091] *)
      ML273 AT %ML273 : ULINT := 16#0123456789ABCDEF;  (* T3D[1092]|T3D[1093]|T3D[1094]|T3D[1095] *)
      ML274 AT %ML274 : ULINT := 16#0123456789ABCDEF;  (* T3D[1096]|T3D[1097]|T3D[1098]|T3D[1099] *)
      ML275 AT %ML275 : ULINT := 16#0123456789ABCDEF;  (* T3D[1100]|T3D[1101]|T3D[1102]|T3D[1103] *)
      ML276 AT %ML276 : ULINT := 16#0123456789ABCDEF;  (* T3D[1104]|T3D[1105]|T3D[1106]|T3D[1107] *)
      ML277 AT %ML277 : ULINT := 16#0123456789ABCDEF;  (* T3D[1108]|T3D[1109]|T3D[1110]|T3D[1111] *)
      ML278 AT %ML278 : ULINT := 16#0123456789ABCDEF;  (* T3D[1112]|T3D[1113]|T3D[1114]|T3D[1115] *)
      ML279 AT %ML279 : ULINT := 16#0123456789ABCDEF;  (* T3D[1116]|T3D[1117]|T3D[1118]|T3D[1119] *)
      ML280 AT %ML280 : ULINT := 16#0123456789ABCDEF;  (* T3D[1120]|T3D[1121]|T3D[1122]|T3D[1123] *)
      ML281 AT %ML281 : ULINT := 16#0123456789ABCDEF;  (* T3D[1124]|T3D[1125]|T3D[1126]|T3D[1127] *)
      ML282 AT %ML282 : ULINT := 16#0123456789ABCDEF;  (* T3D[1128]|T3D[1129]|T3D[1130]|T3D[1131] *)
      ML283 AT %ML283 : ULINT := 16#0123456789ABCDEF;  (* T3D[1132]|T3D[1133]|T3D[1134]|T3D[1135] *)
      ML284 AT %ML284 : ULINT := 16#0123456789ABCDEF;  (* T3D[1136]|T3D[1137]|T3D[1138]|T3D[1139] *)
      ML285 AT %ML285 : ULINT := 16#0123456789ABCDEF;  (* T3D[1140]|T3D[1141]|T3D[1142]|T3D[1143] *)
      ML286 AT %ML286 : ULINT := 16#0123456789ABCDEF;  (* T3D[1144]|T3D[1145]|T3D[1146]|T3D[1147] *)
      ML287 AT %ML287 : ULINT := 16#0123456789ABCDEF;  (* T3D[1148]|T3D[1149]|T3D[1150]|T3D[1151] *)
      ML288 AT %ML288 : ULINT := 16#0123456789ABCDEF;  (* T3D[1152]|T3D[1153]|T3D[1154]|T3D[1155] *)
      ML289 AT %ML289 : ULINT := 16#0123456789ABCDEF;  (* T3D[1156]|T3D[1157]|T3D[1158]|T3D[1159] *)
      ML290 AT %ML290 : ULINT := 16#0123456789ABCDEF;  (* T3D[1160]|T3D[1161]|T3D[1162]|T3D[1163] *)
      ML291 AT %ML291 : ULINT := 16#0123456789ABCDEF;  (* T3D[1164]|T3D[1165]|T3D[1166]|T3D[1167] *)
      ML292 AT %ML292 : ULINT := 16#0123456789ABCDEF;  (* T3D[1168]|T3D[1169]|T3D[1170]|T3D[1171] *)
      ML293 AT %ML293 : ULINT := 16#0123456789ABCDEF;  (* T3D[1172]|T3D[1173]|T3D[1174]|T3D[1175] *)
      ML294 AT %ML294 : ULINT := 16#0123456789ABCDEF;  (* T3D[1176]|T3D[1177]|T3D[1178]|T3D[1179] *)
      ML295 AT %ML295 : ULINT := 16#0123456789ABCDEF;  (* T3D[1180]|T3D[1181]|T3D[1182]|T3D[1183] *)
      ML296 AT %ML296 : ULINT := 16#0123456789ABCDEF;  (* T3D[1184]|T3D[1185]|T3D[1186]|T3D[1187] *)
      ML297 AT %ML297 : ULINT := 16#0123456789ABCDEF;  (* T3D[1188]|T3D[1189]|T3D[1190]|T3D[1191] *)
      ML298 AT %ML298 : ULINT := 16#0123456789ABCDEF;  (* T3D[1192]|T3D[1193]|T3D[1194]|T3D[1195] *)
      ML299 AT %ML299 : ULINT := 16#0123456789ABCDEF;  (* T3D[1196]|T3D[1197]|T3D[1198]|T3D[1199] *)
      ML300 AT %ML300 : ULINT := 16#0123456789ABCDEF;  (* T3D[1200]|T3D[1201]|T3D[1202]|T3D[1203] *)
      ML301 AT %ML301 : ULINT := 16#0123456789ABCDEF;  (* T3D[1204]|T3D[1205]|T3D[1206]|T3D[1207] *)
      ML302 AT %ML302 : ULINT := 16#0123456789ABCDEF;  (* T3D[1208]|T3D[1209]|T3D[1210]|T3D[1211] *)
      ML303 AT %ML303 : ULINT := 16#0123456789ABCDEF;  (* T3D[1212]|T3D[1213]|T3D[1214]|T3D[1215] *)
      ML304 AT %ML304 : ULINT := 16#0123456789ABCDEF;  (* T3D[1216]|T3D[1217]|T3D[1218]|T3D[1219] *)
      ML305 AT %ML305 : ULINT := 16#0123456789ABCDEF;  (* T3D[1220]|T3D[1221]|T3D[1222]|T3D[1223] *)
      ML306 AT %ML306 : ULINT := 16#0123456789ABCDEF;  (* T3D[1224]|T3D[1225]|T3D[1226]|T3D[1227] *)
      ML307 AT %ML307 : ULINT := 16#0123456789ABCDEF;  (* T3D[1228]|T3D[1229]|T3D[1230]|T3D[1231] *)
      ML308 AT %ML308 : ULINT := 16#0123456789ABCDEF;  (* T3D[1232]|T3D[1233]|T3D[1234]|T3D[1235] *)
      ML309 AT %ML309 : ULINT := 16#0123456789ABCDEF;  (* T3D[1236]|T3D[1237]|T3D[1238]|T3D[1239] *)
      ML310 AT %ML310 : ULINT := 16#0123456789ABCDEF;  (* T3D[1240]|T3D[1241]|T3D[1242]|T3D[1243] *)
      ML311 AT %ML311 : ULINT := 16#0123456789ABCDEF;  (* T3D[1244]|T3D[1245]|T3D[1246]|T3D[1247] *)
      ML312 AT %ML312 : ULINT := 16#0123456789ABCDEF;  (* T3D[1248]|T3D[1249]|T3D[1250]|T3D[1251] *)
      ML313 AT %ML313 : ULINT := 16#0123456789ABCDEF;  (* T3D[1252]|T3D[1253]|T3D[1254]|T3D[1255] *)
      ML314 AT %ML314 : ULINT := 16#0123456789ABCDEF;  (* T3D[1256]|T3D[1257]|T3D[1258]|T3D[1259] *)
      ML315 AT %ML315 : ULINT := 16#0123456789ABCDEF;  (* T3D[1260]|T3D[1261]|T3D[1262]|T3D[1263] *)
      ML316 AT %ML316 : ULINT := 16#0123456789ABCDEF;  (* T3D[1264]|T3D[1265]|T3D[1266]|T3D[1267] *)
      ML317 AT %ML317 : ULINT := 16#0123456789ABCDEF;  (* T3D[1268]|T3D[1269]|T3D[1270]|T3D[1271] *)
      ML318 AT %ML318 : ULINT := 16#0123456789ABCDEF;  (* T3D[1272]|T3D[1273]|T3D[1274]|T3D[1275] *)
      ML319 AT %ML319 : ULINT := 16#0123456789ABCDEF;  (* T3D[1276]|T3D[1277]|T3D[1278]|T3D[1279] *)
      ML320 AT %ML320 : ULINT := 16#0123456789ABCDEF;  (* T3D[1280]|T3D[1281]|T3D[1282]|T3D[1283] *)
      ML321 AT %ML321 : ULINT := 16#0123456789ABCDEF;  (* T3D[1284]|T3D[1285]|T3D[1286]|T3D[1287] *)
      ML322 AT %ML322 : ULINT := 16#0123456789ABCDEF;  (* T3D[1288]|T3D[1289]|T3D[1290]|T3D[1291] *)
      ML323 AT %ML323 : ULINT := 16#0123456789ABCDEF;  (* T3D[1292]|T3D[1293]|T3D[1294]|T3D[1295] *)
      ML324 AT %ML324 : ULINT := 16#0123456789ABCDEF;  (* T3D[1296]|T3D[1297]|T3D[1298]|T3D[1299] *)
      ML325 AT %ML325 : ULINT := 16#0123456789ABCDEF;  (* T3D[1300]|T3D[1301]|T3D[1302]|T3D[1303] *)
      ML326 AT %ML326 : ULINT := 16#0123456789ABCDEF;  (* T3D[1304]|T3D[1305]|T3D[1306]|T3D[1307] *)
      ML327 AT %ML327 : ULINT := 16#0123456789ABCDEF;  (* T3D[1308]|T3D[1309]|T3D[1310]|T3D[1311] *)
      ML328 AT %ML328 : ULINT := 16#0123456789ABCDEF;  (* T3D[1312]|T3D[1313]|T3D[1314]|T3D[1315] *)
      ML329 AT %ML329 : ULINT := 16#0123456789ABCDEF;  (* T3D[1316]|T3D[1317]|T3D[1318]|T3D[1319] *)
      ML330 AT %ML330 : ULINT := 16#0123456789ABCDEF;  (* T3D[1320]|T3D[1321]|T3D[1322]|T3D[1323] *)
      ML331 AT %ML331 : ULINT := 16#0123456789ABCDEF;  (* T3D[1324]|T3D[1325]|T3D[1326]|T3D[1327] *)
      ML332 AT %ML332 : ULINT := 16#0123456789ABCDEF;  (* T3D[1328]|T3D[1329]|T3D[1330]|T3D[1331] *)
      ML333 AT %ML333 : ULINT := 16#0123456789ABCDEF;  (* T3D[1332]|T3D[1333]|T3D[1334]|T3D[1335] *)
      ML334 AT %ML334 : ULINT := 16#0123456789ABCDEF;  (* T3D[1336]|T3D[1337]|T3D[1338]|T3D[1339] *)
      ML335 AT %ML335 : ULINT := 16#0123456789ABCDEF;  (* T3D[1340]|T3D[1341]|T3D[1342]|T3D[1343] *)
      ML336 AT %ML336 : ULINT := 16#0123456789ABCDEF;  (* T3D[1344]|T3D[1345]|T3D[1346]|T3D[1347] *)
      ML337 AT %ML337 : ULINT := 16#0123456789ABCDEF;  (* T3D[1348]|T3D[1349]|T3D[1350]|T3D[1351] *)
      ML338 AT %ML338 : ULINT := 16#0123456789ABCDEF;  (* T3D[1352]|T3D[1353]|T3D[1354]|T3D[1355] *)
      ML339 AT %ML339 : ULINT := 16#0123456789ABCDEF;  (* T3D[1356]|T3D[1357]|T3D[1358]|T3D[1359] *)
      ML340 AT %ML340 : ULINT := 16#0123456789ABCDEF;  (* T3D[1360]|T3D[1361]|T3D[1362]|T3D[1363] *)
      ML341 AT %ML341 : ULINT := 16#0123456789ABCDEF;  (* T3D[1364]|T3D[1365]|T3D[1366]|T3D[1367] *)
      ML342 AT %ML342 : ULINT := 16#0123456789ABCDEF;  (* T3D[1368]|T3D[1369]|T3D[1370]|T3D[1371] *)
      ML343 AT %ML343 : ULINT := 16#0123456789ABCDEF;  (* T3D[1372]|T3D[1373]|T3D[1374]|T3D[1375] *)
      ML344 AT %ML344 : ULINT := 16#0123456789ABCDEF;  (* T3D[1376]|T3D[1377]|T3D[1378]|T3D[1379] *)
      ML345 AT %ML345 : ULINT := 16#0123456789ABCDEF;  (* T3D[1380]|T3D[1381]|T3D[1382]|T3D[1383] *)
      ML346 AT %ML346 : ULINT := 16#0123456789ABCDEF;  (* T3D[1384]|T3D[1385]|T3D[1386]|T3D[1387] *)
      ML347 AT %ML347 : ULINT := 16#0123456789ABCDEF;  (* T3D[1388]|T3D[1389]|T3D[1390]|T3D[1391] *)
      ML348 AT %ML348 : ULINT := 16#0123456789ABCDEF;  (* T3D[1392]|T3D[1393]|T3D[1394]|T3D[1395] *)
      ML349 AT %ML349 : ULINT := 16#0123456789ABCDEF;  (* T3D[1396]|T3D[1397]|T3D[1398]|T3D[1399] *)
      ML350 AT %ML350 : ULINT := 16#0123456789ABCDEF;  (* T3D[1400]|T3D[1401]|T3D[1402]|T3D[1403] *)
      ML351 AT %ML351 : ULINT := 16#0123456789ABCDEF;  (* T3D[1404]|T3D[1405]|T3D[1406]|T3D[1407] *)
      ML352 AT %ML352 : ULINT := 16#0123456789ABCDEF;  (* T3D[1408]|T3D[1409]|T3D[1410]|T3D[1411] *)
      ML353 AT %ML353 : ULINT := 16#0123456789ABCDEF;  (* T3D[1412]|T3D[1413]|T3D[1414]|T3D[1415] *)
      ML354 AT %ML354 : ULINT := 16#0123456789ABCDEF;  (* T3D[1416]|T3D[1417]|T3D[1418]|T3D[1419] *)
